LIN {X 0,Y 236.91,Z 434.305,A -85,B 0,C 180,E1 -22367.058,E2 -22367.058} C_VEL
LIN {X 0,Y 236.461,Z 436.627,A -85,B 0,C 180,E1 -22367.156,E2 -22367.156} C_VEL
LIN {X 0,Y 234.937,Z 442.325,A -85,B 0,C 180,E1 -22367.31,E2 -22367.31} C_VEL
LIN {X 0,Y 231.156,Z 451.531,A -85,B 0,C 180,E1 -22367.278,E2 -22367.278} C_VEL
LIN {X 0,Y 226.925,Z 460.5,A -85,B 0,C 180,E1 -22367.362,E2 -22367.362} C_VEL
LIN {X 0,Y 224.696,Z 465.695,A -85,B 0,C 180,E1 -22367.708,E2 -22367.708} C_VEL
LIN {X 0,Y 219.819,Z 477.382,A -85,B 0,C 180,E1 -22369.057,E2 -22369.057} C_VEL
LIN {X 0,Y 214.094,Z 488.851,A -85,B 0,C 180,E1 -22370.817,E2 -22370.817} C_VEL
LIN {X 0,Y 208.781,Z 498.232,A -85,B 0,C 180,E1 -22372.714,E2 -22372.714} C_VEL
LIN {X 0,Y 202.847,Z 507.555,A -85,B 0,C 180,E1 -22375.141,E2 -22375.141} C_VEL
LIN {X 0,Y 197.376,Z 515.201,A -85,B 0,C 180,E1 -22377.724,E2 -22377.724} C_VEL
LIN {X 0,Y 192.63,Z 521.438,A -85,B 0,C 180,E1 -22380.499,E2 -22380.499} C_VEL
LIN {X 0,Y 188.329,Z 526.526,A -85,B 0,C 180,E1 -22383.403,E2 -22383.403} C_VEL
LIN {X 0,Y 184.743,Z 530.596,A -85,B 0,C 180,E1 -22386.463,E2 -22386.463} C_VEL
LIN {X 0,Y 181.766,Z 533.709,A -85,B 0,C 180,E1 -22389.642,E2 -22389.642} C_VEL
LIN {X 0,Y 178.613,Z 536.431,A -85,B 0,C 180,E1 -22394.018,E2 -22394.018} C_VEL
LIN {X 0,Y 176.91,Z 537.692,A -85,B 0,C 180,E1 -22398.548,E2 -22398.548} C_VEL
LIN {X 0,Y 176.292,Z 537.397,A -85,B 0,C 180,E1 -22403.136,E2 -22403.136} C_VEL
LIN {X 0,Y 176.352,Z 536.677,A -85,B 0,C 180,E1 -22405.433,E2 -22405.433} C_VEL
LIN {X 0,Y 176.44,Z 535.538,A -85,B 0,C 180,E1 -22407.721,E2 -22407.721} C_VEL
LIN {X 0,Y 176.671,Z 533.977,A -85,B 0,C 180,E1 -22410.004,E2 -22410.004} C_VEL
LIN {X 0,Y 176.674,Z 530.644,A -85,B 0,C 180,E1 -22413.424,E2 -22413.424} C_VEL
LIN {X 0,Y 176.697,Z 527.213,A -85,B 0,C 180,E1 -22416.079,E2 -22416.079} C_VEL
LIN {X 0,Y 176.947,Z 521.277,A -85,B 0,C 180,E1 -22419.721,E2 -22419.721} C_VEL
LIN {X 0,Y 177.588,Z 514.102,A -85,B 0,C 180,E1 -22423.155,E2 -22423.155} C_VEL
LIN {X 0,Y 178.93,Z 505.14,A -85,B 0,C 180,E1 -22426.547,E2 -22426.547} C_VEL
LIN {X 0,Y 180.296,Z 495.891,A -85,B 0,C 180,E1 -22429.351,E2 -22429.351} C_VEL
LIN {X 0,Y 181.95,Z 485.894,A -85,B 0,C 180,E1 -22431.782,E2 -22431.782} C_VEL
LIN {X 0,Y 183.735,Z 474.492,A -85,B 0,C 180,E1 -22433.981,E2 -22433.981} C_VEL
LIN {X 0,Y 185.536,Z 462.13,A -85,B 0,C 180,E1 -22435.825,E2 -22435.825} C_VEL
LIN {X 0,Y 187.111,Z 449.244,A -85,B 0,C 180,E1 -22437.244,E2 -22437.244} C_VEL
LIN {X 0,Y 188.205,Z 437.063,A -85,B 0,C 180,E1 -22438.205,E2 -22438.205} C_VEL
LIN {X 0,Y 190.833,Z 387.8,A -85,B 0,C 180,E1 -22440.716,E2 -22440.716} C_VEL
LIN {X 0,Y 187.268,Z 349.514,A -85,B 0,C 180,E1 -22443.19,E2 -22443.19} C_VEL
LIN {X 0,Y 180.421,Z 327.475,A -85,B 0,C 180,E1 -22445.255,E2 -22445.255} C_VEL
LIN {X 0,Y 178.472,Z 318.252,A -85,B 0,C 180,E1 -22449.876,E2 -22449.876} C_VEL
LIN {X 0,Y 178.39,Z 318.26,A -85,B 0,C 180,E1 -22455.164,E2 -22455.164} C_VEL
LIN {X 0,Y 178.395,Z 318.261,A -85,B 0,C 180,E1 -22458.461,E2 -22458.461} C_VEL
LIN {X 0,Y 178.416,Z 318.259,A -85,B 0,C 180,E1 -22463.78,E2 -22463.78} C_VEL
LIN {X 0,Y 178.479,Z 318.252,A -85,B 0,C 180,E1 -22466.544,E2 -22466.544} C_VEL
LIN {X 0,Y 178.426,Z 318.258,A -85,B 0,C 180,E1 -22471.791,E2 -22471.791} C_VEL
LIN {X 0,Y 178.512,Z 318.249,A -85,B 0,C 180,E1 -22474.888,E2 -22474.888} C_VEL
LIN {X 0,Y 178.6,Z 318.237,A -85,B 0,C 180,E1 -22481.65,E2 -22481.65} C_VEL
LIN {X 0,Y 178.627,Z 318.23,A -85,B 0,C 180,E1 -22486.344,E2 -22486.344} C_VEL
LIN {X 0,Y 178.897,Z 318.2,A -85,B 0,C 180,E1 -22490.958,E2 -22490.958} C_VEL
LIN {X 0,Y 179.133,Z 318.171,A -85,B 0,C 180,E1 -22497.75,E2 -22497.75} C_VEL
LIN {X 0,Y 179.35,Z 318.142,A -85,B 0,C 180,E1 -22499.999,E2 -22499.999} C_VEL
LIN {X 0,Y 178.839,Z 318.205,A -85,B 0,C 180,E1 -22504.507,E2 -22504.507} C_VEL
LIN {X 0,Y 178.896,Z 318.199,A -85,B 0,C 180,E1 -22509.04,E2 -22509.04} C_VEL
LIN {X 0,Y 178.627,Z 318.235,A -85,B 0,C 180,E1 -22513.653,E2 -22513.653} C_VEL
LIN {X 0,Y 178.545,Z 318.239,A -85,B 0,C 180,E1 -22519.149,E2 -22519.149} C_VEL
LIN {X 0,Y 178.513,Z 318.247,A -85,B 0,C 180,E1 -22525.113,E2 -22525.113} C_VEL
LIN {X 0,Y 178.515,Z 318.249,A -85,B 0,C 180,E1 -22529.992,E2 -22529.992} C_VEL
LIN {X 0,Y 178.478,Z 318.25,A -85,B 0,C 180,E1 -22534.218,E2 -22534.218} C_VEL
LIN {X 0,Y 178.39,Z 318.262,A -85,B 0,C 180,E1 -22539.074,E2 -22539.074} C_VEL
LIN {X 0,Y 178.404,Z 318.261,A -85,B 0,C 180,E1 -22542.042,E2 -22542.042} C_VEL
LIN {X 0,Y 178.426,Z 318.254,A -85,B 0,C 180,E1 -22545.152,E2 -22545.152} C_VEL
LIN {X 0,Y 178.448,Z 318.257,A -85,B 0,C 180,E1 -22548.441,E2 -22548.441} C_VEL
LIN {X 0,Y 178.487,Z 318.249,A -85,B 0,C 180,E1 -22551.951,E2 -22551.951} C_VEL
LIN {X 0,Y 178.487,Z 318.252,A -85,B 0,C 180,E1 -22556.546,E2 -22556.546} C_VEL
LIN {X 0,Y 178.52,Z 318.246,A -85,B 0,C 180,E1 -22560.006,E2 -22560.006} C_VEL
LIN {X 0,Y 178.523,Z 318.247,A -85,B 0,C 180,E1 -22564.881,E2 -22564.881} C_VEL
LIN {X 0,Y 178.622,Z 318.233,A -85,B 0,C 180,E1 -22570.782,E2 -22570.782} C_VEL
LIN {X 0,Y 178.665,Z 318.228,A -85,B 0,C 180,E1 -22576.346,E2 -22576.346} C_VEL
LIN {X 0,Y 178.977,Z 318.19,A -85,B 0,C 180,E1 -22580.96,E2 -22580.96} C_VEL
LIN {X 0,Y 179.152,Z 318.165,A -85,B 0,C 180,E1 -22587.748,E2 -22587.748} C_VEL
LIN {X 0,Y 179.368,Z 318.141,A -85,B 0,C 180,E1 -22589.996,E2 -22589.996} C_VEL
LIN {X 0,Y 178.872,Z 318.201,A -85,B 0,C 180,E1 -22594.503,E2 -22594.503} C_VEL
LIN {X 0,Y 178.97,Z 318.192,A -85,B 0,C 180,E1 -22599.033,E2 -22599.033} C_VEL
LIN {X 0,Y 178.684,Z 318.226,A -85,B 0,C 180,E1 -22603.645,E2 -22603.645} C_VEL
LIN {X 0,Y 178.674,Z 318.227,A -85,B 0,C 180,E1 -22608.335,E2 -22608.335} C_VEL
LIN {X 0,Y 178.522,Z 318.248,A -85,B 0,C 180,E1 -22613.177,E2 -22613.177} C_VEL
LIN {X 0,Y 178.512,Z 318.249,A -85,B 0,C 180,E1 -22617.309,E2 -22617.309} C_VEL
LIN {X 0,Y 181.026,Z 325.006,A -85,B 0,C 180,E1 -22618.016,E2 -22618.016} C_VEL
LIN {X 0,Y 191.33,Z 351.912,A -85,B 0,C 180,E1 -22620.639,E2 -22620.639} C_VEL
LIN {X 0,Y 192.125,Z 354.048,A -85,B 0,C 180,E1 -22620.836,E2 -22620.836} C_VEL
LIN {X 0,Y 188.406,Z 416.37,A -85,B 0,C 180,E1 -22623.942,E2 -22623.942} C_VEL
LIN {X 0,Y 187.548,Z 428.759,A -85,B 0,C 180,E1 -22624.945,E2 -22624.945} C_VEL
LIN {X 0,Y 186.105,Z 441.894,A -85,B 0,C 180,E1 -22626.408,E2 -22626.408} C_VEL
LIN {X 0,Y 184.486,Z 453.979,A -85,B 0,C 180,E1 -22628.215,E2 -22628.215} C_VEL
LIN {X 0,Y 182.727,Z 466.025,A -85,B 0,C 180,E1 -22630.525,E2 -22630.525} C_VEL
LIN {X 0,Y 181.01,Z 476.642,A -85,B 0,C 180,E1 -22633.113,E2 -22633.113} C_VEL
LIN {X 0,Y 179.505,Z 486.117,A -85,B 0,C 180,E1 -22635.979,E2 -22635.979} C_VEL
LIN {X 0,Y 178.24,Z 494.278,A -85,B 0,C 180,E1 -22639.015,E2 -22639.015} C_VEL
LIN {X 0,Y 177.173,Z 501.741,A -85,B 0,C 180,E1 -22642.486,E2 -22642.486} C_VEL
LIN {X 0,Y 176.5,Z 507.92,A -85,B 0,C 180,E1 -22646.121,E2 -22646.121} C_VEL
LIN {X 0,Y 176.054,Z 513.063,A -85,B 0,C 180,E1 -22650.068,E2 -22650.068} C_VEL
LIN {X 0,Y 176.088,Z 516.711,A -85,B 0,C 180,E1 -22653.959,E2 -22653.959} C_VEL
LIN {X 0,Y 176.507,Z 518.42,A -85,B 0,C 180,E1 -22656.537,E2 -22656.537} C_VEL
LIN {X 0,Y 177.134,Z 519.648,A -85,B 0,C 180,E1 -22659.08,E2 -22659.08} C_VEL
LIN {X 0,Y 178.046,Z 520.342,A -85,B 0,C 180,E1 -22661.593,E2 -22661.593} C_VEL
LIN {X 0,Y 179.227,Z 520.555,A -85,B 0,C 180,E1 -22664.07,E2 -22664.07} C_VEL
LIN {X 0,Y 180.699,Z 520.318,A -85,B 0,C 180,E1 -22666.506,E2 -22666.506} C_VEL
LIN {X 0,Y 182.451,Z 519.566,A -85,B 0,C 180,E1 -22668.897,E2 -22668.897} C_VEL
LIN {X 0,Y 184.712,Z 518.19,A -85,B 0,C 180,E1 -22671.532,E2 -22671.532} C_VEL
LIN {X 0,Y 187.992,Z 515.646,A -85,B 0,C 180,E1 -22674.638,E2 -22674.638} C_VEL
LIN {X 0,Y 192.28,Z 511.728,A -85,B 0,C 180,E1 -22677.906,E2 -22677.906} C_VEL
LIN {X 0,Y 197.278,Z 506.305,A -85,B 0,C 180,E1 -22681.163,E2 -22681.163} C_VEL
LIN {X 0,Y 202.461,Z 499.893,A -85,B 0,C 180,E1 -22683.982,E2 -22683.982} C_VEL
LIN {X 0,Y 208.425,Z 491.476,A -85,B 0,C 180,E1 -22686.779,E2 -22686.779} C_VEL
LIN {X 0,Y 214.293,Z 481.83,A -85,B 0,C 180,E1 -22689.211,E2 -22689.211} C_VEL
LIN {X 0,Y 219.321,Z 472.21,A -85,B 0,C 180,E1 -22691.086,E2 -22691.086} C_VEL
LIN {X 0,Y 224.023,Z 461.664,A -85,B 0,C 180,E1 -22692.687,E2 -22692.687} C_VEL
LIN {X 0,Y 228.213,Z 450.32,A -85,B 0,C 180,E1 -22694.037,E2 -22694.037} C_VEL
LIN {X 0,Y 231.893,Z 438.008,A -85,B 0,C 180,E1 -22695.155,E2 -22695.155} C_VEL
LIN {X 0,Y 234.808,Z 424.844,A -85,B 0,C 180,E1 -22696.021,E2 -22696.021} C_VEL
LIN {X 0,Y 237.683,Z 405.575,A -85,B 0,C 180,E1 -22696.846,E2 -22696.846} C_VEL
LIN {X 0,Y 239.653,Z 391.45,A -85,B 0,C 180,E1 -22697.393,E2 -22697.393} C_VEL
LIN {X 0,Y 236.976,Z 385.819,A -85,B 0,C 180,E1 -22700.059,E2 -22700.059} C_VEL
LIN {X 0,Y 235.295,Z 382.982,A -85,B 0,C 180,E1 -22702.06,E2 -22702.06} C_VEL
LIN {X 0,Y 234.145,Z 380.911,A -85,B 0,C 180,E1 -22703.778,E2 -22703.778} C_VEL
LIN {X 0,Y 232.449,Z 378.806,A -85,B 0,C 180,E1 -22707.56,E2 -22707.56} C_VEL
LIN {X 0,Y 232.17,Z 378.586,A -85,B 0,C 180,E1 -22708.97,E2 -22708.97} C_VEL
LIN {X 0,Y 232.07,Z 379.141,A -85,B 0,C 180,E1 -22712.025,E2 -22712.025} C_VEL
LIN {X 0,Y 232.263,Z 379.966,A -85,B 0,C 180,E1 -22713.548,E2 -22713.548} C_VEL
LIN {X 0,Y 233.683,Z 384.466,A -85,B 0,C 180,E1 -22717.461,E2 -22717.461} C_VEL
LIN {X 0,Y 235.599,Z 389.873,A -85,B 0,C 180,E1 -22720.459,E2 -22720.459} C_VEL
LIN {X 0,Y 237.273,Z 395.332,A -85,B 0,C 180,E1 -22722.542,E2 -22722.542} C_VEL
LIN {X 0,Y 238.737,Z 400.557,A -85,B 0,C 180,E1 -22724.133,E2 -22724.133} C_VEL
LIN {X 0,Y 234.037,Z 433.293,A -85,B 0,C 180,E1 -22725.453,E2 -22725.453} C_VEL
LIN {X 0,Y 231.248,Z 445.622,A -85,B 0,C 180,E1 -22726.117,E2 -22726.117} C_VEL
LIN {X 0,Y 227.754,Z 457.295,A -85,B 0,C 180,E1 -22726.952,E2 -22726.952} C_VEL
LIN {X 0,Y 224.696,Z 465.695,A -85,B 0,C 180,E1 -22727.708,E2 -22727.708} C_VEL
LIN {X 0,Y 222.306,Z 470.885,A -85,B 0,C 180,E1 -22728.108,E2 -22728.108} C_VEL
LIN {X 0,Y 217.101,Z 479.22,A -85,B 0,C 180,E1 -22728.492,E2 -22728.492} C_VEL
LIN {X 0,Y 211.532,Z 487.12,A -85,B 0,C 180,E1 -22729.028,E2 -22729.028} C_VEL
LIN {X 0,Y 208.601,Z 491.616,A -85,B 0,C 180,E1 -22729.68,E2 -22729.68} C_VEL
LIN {X 0,Y 202.28,Z 501.788,A -85,B 0,C 180,E1 -22731.933,E2 -22731.933} C_VEL
LIN {X 0,Y 196.179,Z 510.356,A -85,B 0,C 180,E1 -22734.406,E2 -22734.406} C_VEL
LIN {X 0,Y 189.822,Z 518.369,A -85,B 0,C 180,E1 -22737.538,E2 -22737.538} C_VEL
LIN {X 0,Y 184.917,Z 523.953,A -85,B 0,C 180,E1 -22740.398,E2 -22740.398} C_VEL
LIN {X 0,Y 180.649,Z 528.482,A -85,B 0,C 180,E1 -22743.485,E2 -22743.485} C_VEL
LIN {X 0,Y 177.137,Z 531.918,A -85,B 0,C 180,E1 -22746.631,E2 -22746.631} C_VEL
LIN {X 0,Y 173.311,Z 535.193,A -85,B 0,C 180,E1 -22751.076,E2 -22751.076} C_VEL
LIN {X 0,Y 171.784,Z 536.265,A -85,B 0,C 180,E1 -22753.364,E2 -22753.364} C_VEL
LIN {X 0,Y 169.936,Z 537.251,A -85,B 0,C 180,E1 -22758.071,E2 -22758.071} C_VEL
LIN {X 0,Y 169.256,Z 536.745,A -85,B 0,C 180,E1 -22762.849,E2 -22762.849} C_VEL
LIN {X 0,Y 169.298,Z 535.932,A -85,B 0,C 180,E1 -22765.242,E2 -22765.242} C_VEL
LIN {X 0,Y 169.388,Z 534.689,A -85,B 0,C 180,E1 -22767.626,E2 -22767.626} C_VEL
LIN {X 0,Y 169.653,Z 532.994,A -85,B 0,C 180,E1 -22770.004,E2 -22770.004} C_VEL
LIN {X 0,Y 169.65,Z 529.491,A -85,B 0,C 180,E1 -22773.566,E2 -22773.566} C_VEL
LIN {X 0,Y 169.683,Z 524.72,A -85,B 0,C 180,E1 -22777.141,E2 -22777.141} C_VEL
LIN {X 0,Y 170.031,Z 518.573,A -85,B 0,C 180,E1 -22780.722,E2 -22780.722} C_VEL
LIN {X 0,Y 170.91,Z 510.862,A -85,B 0,C 180,E1 -22784.286,E2 -22784.286} C_VEL
LIN {X 0,Y 172.375,Z 501.133,A -85,B 0,C 180,E1 -22787.808,E2 -22787.808} C_VEL
LIN {X 0,Y 174.04,Z 491.112,A -85,B 0,C 180,E1 -22790.693,E2 -22790.693} C_VEL
LIN {X 0,Y 175.831,Z 480.218,A -85,B 0,C 180,E1 -22793.171,E2 -22793.171} C_VEL
LIN {X 0,Y 177.528,Z 469.019,A -85,B 0,C 180,E1 -22795.188,E2 -22795.188} C_VEL
LIN {X 0,Y 179.35,Z 456.267,A -85,B 0,C 180,E1 -22796.943,E2 -22796.943} C_VEL
LIN {X 0,Y 180.901,Z 442.079,A -85,B 0,C 180,E1 -22798.341,E2 -22798.341} C_VEL
LIN {X 0,Y 181.859,Z 427.344,A -85,B 0,C 180,E1 -22799.283,E2 -22799.283} C_VEL
LIN {X 0,Y 184.052,Z 388.689,A -85,B 0,C 180,E1 -22801.298,E2 -22801.298} C_VEL
LIN {X 0,Y 180.728,Z 351.595,A -85,B 0,C 180,E1 -22803.762,E2 -22803.762} C_VEL
LIN {X 0,Y 173.088,Z 327.033,A -85,B 0,C 180,E1 -22806.198,E2 -22806.198} C_VEL
LIN {X 0,Y 171.422,Z 319.131,A -85,B 0,C 180,E1 -22810.414,E2 -22810.414} C_VEL
LIN {X 0,Y 171.317,Z 319.139,A -85,B 0,C 180,E1 -22815.78,E2 -22815.78} C_VEL
LIN {X 0,Y 171.341,Z 319.141,A -85,B 0,C 180,E1 -22821.198,E2 -22821.198} C_VEL
LIN {X 0,Y 171.396,Z 319.136,A -85,B 0,C 180,E1 -22825.092,E2 -22825.092} C_VEL
LIN {X 0,Y 171.391,Z 319.135,A -85,B 0,C 180,E1 -22830.522,E2 -22830.522} C_VEL
LIN {X 0,Y 171.431,Z 319.126,A -85,B 0,C 180,E1 -22835.796,E2 -22835.796} C_VEL
LIN {X 0,Y 171.501,Z 319.122,A -85,B 0,C 180,E1 -22840.861,E2 -22840.861} C_VEL
LIN {X 0,Y 171.542,Z 319.113,A -85,B 0,C 180,E1 -22845.769,E2 -22845.769} C_VEL
LIN {X 0,Y 171.836,Z 319.079,A -85,B 0,C 180,E1 -22850.583,E2 -22850.583} C_VEL
LIN {X 0,Y 171.79,Z 319.083,A -85,B 0,C 180,E1 -22855.306,E2 -22855.306} C_VEL
LIN {X 0,Y 172.314,Z 319.018,A -85,B 0,C 180,E1 -22859.999,E2 -22859.999} C_VEL
LIN {X 0,Y 171.788,Z 319.084,A -85,B 0,C 180,E1 -22864.692,E2 -22864.692} C_VEL
LIN {X 0,Y 171.834,Z 319.078,A -85,B 0,C 180,E1 -22869.415,E2 -22869.415} C_VEL
LIN {X 0,Y 171.541,Z 319.116,A -85,B 0,C 180,E1 -22874.229,E2 -22874.229} C_VEL
LIN {X 0,Y 171.471,Z 319.121,A -85,B 0,C 180,E1 -22879.497,E2 -22879.497} C_VEL
LIN {X 0,Y 171.451,Z 319.128,A -85,B 0,C 180,E1 -22885.607,E2 -22885.607} C_VEL
LIN {X 0,Y 171.434,Z 319.129,A -85,B 0,C 180,E1 -22890.584,E2 -22890.584} C_VEL
LIN {X 0,Y 171.388,Z 319.132,A -85,B 0,C 180,E1 -22895.034,E2 -22895.034} C_VEL
LIN {X 0,Y 171.352,Z 319.139,A -85,B 0,C 180,E1 -22898.806,E2 -22898.806} C_VEL
LIN {X 0,Y 171.341,Z 319.138,A -85,B 0,C 180,E1 -22904.209,E2 -22904.209} C_VEL
LIN {X 0,Y 171.38,Z 319.136,A -85,B 0,C 180,E1 -22908.994,E2 -22908.994} C_VEL
LIN {X 0,Y 171.434,Z 319.127,A -85,B 0,C 180,E1 -22912.053,E2 -22912.053} C_VEL
LIN {X 0,Y 171.416,Z 319.132,A -85,B 0,C 180,E1 -22917.791,E2 -22917.791} C_VEL
LIN {X 0,Y 171.446,Z 319.124,A -85,B 0,C 180,E1 -22920.533,E2 -22920.533} C_VEL
LIN {X 0,Y 171.452,Z 319.128,A -85,B 0,C 180,E1 -22925.799,E2 -22925.799} C_VEL
LIN {X 0,Y 171.578,Z 319.11,A -85,B 0,C 180,E1 -22930.87,E2 -22930.87} C_VEL
LIN {X 0,Y 171.581,Z 319.11,A -85,B 0,C 180,E1 -22935.771,E2 -22935.771} C_VEL
LIN {X 0,Y 171.903,Z 319.072,A -85,B 0,C 180,E1 -22940.585,E2 -22940.585} C_VEL
LIN {X 0,Y 171.823,Z 319.077,A -85,B 0,C 180,E1 -22945.304,E2 -22945.304} C_VEL
LIN {X 0,Y 172.331,Z 319.017,A -85,B 0,C 180,E1 -22949.996,E2 -22949.996} C_VEL
LIN {X 0,Y 171.821,Z 319.079,A -85,B 0,C 180,E1 -22954.688,E2 -22954.688} C_VEL
LIN {X 0,Y 171.903,Z 319.071,A -85,B 0,C 180,E1 -22959.407,E2 -22959.407} C_VEL
LIN {X 0,Y 171.609,Z 319.108,A -85,B 0,C 180,E1 -22964.219,E2 -22964.219} C_VEL
LIN {X 0,Y 171.568,Z 319.115,A -85,B 0,C 180,E1 -22969.587,E2 -22969.587} C_VEL
LIN {X 0,Y 171.458,Z 319.126,A -85,B 0,C 180,E1 -22976.082,E2 -22976.082} C_VEL
LIN {X 0,Y 171.471,Z 319.125,A -85,B 0,C 180,E1 -22976.435,E2 -22976.435} C_VEL
LIN {X 0,Y 173.945,Z 325.721,A -85,B 0,C 180,E1 -22977.198,E2 -22977.198} C_VEL
LIN {X 0,Y 184.799,Z 354.048,A -85,B 0,C 180,E1 -22980.101,E2 -22980.101} C_VEL
LIN {X 0,Y 185.267,Z 355.43,A -85,B 0,C 180,E1 -22980.227,E2 -22980.227} C_VEL
LIN {X 0,Y 181.522,Z 416.426,A -85,B 0,C 180,E1 -22983.403,E2 -22983.403} C_VEL
LIN {X 0,Y 180.597,Z 429.111,A -85,B 0,C 180,E1 -22984.462,E2 -22984.462} C_VEL
LIN {X 0,Y 179.185,Z 441.892,A -85,B 0,C 180,E1 -22985.932,E2 -22985.932} C_VEL
LIN {X 0,Y 177.61,Z 453.393,A -85,B 0,C 180,E1 -22987.686,E2 -22987.686} C_VEL
LIN {X 0,Y 175.785,Z 465.628,A -85,B 0,C 180,E1 -22990.084,E2 -22990.084} C_VEL
LIN {X 0,Y 174.131,Z 475.694,A -85,B 0,C 180,E1 -22992.561,E2 -22992.561} C_VEL
LIN {X 0,Y 172.449,Z 485.991,A -85,B 0,C 180,E1 -22995.742,E2 -22995.742} C_VEL
LIN {X 0,Y 171.127,Z 494.299,A -85,B 0,C 180,E1 -22998.922,E2 -22998.922} C_VEL
LIN {X 0,Y 170.077,Z 501.686,A -85,B 0,C 180,E1 -23002.448,E2 -23002.448} C_VEL
LIN {X 0,Y 169.42,Z 507.657,A -85,B 0,C 180,E1 -23006.048,E2 -23006.048} C_VEL
LIN {X 0,Y 168.958,Z 512.818,A -85,B 0,C 180,E1 -23010.057,E2 -23010.057} C_VEL
LIN {X 0,Y 169,Z 516.675,A -85,B 0,C 180,E1 -23014.111,E2 -23014.111} C_VEL
LIN {X 0,Y 169.734,Z 519.274,A -85,B 0,C 180,E1 -23018.122,E2 -23018.122} C_VEL
LIN {X 0,Y 170.736,Z 520.456,A -85,B 0,C 180,E1 -23021.188,E2 -23021.188} C_VEL
LIN {X 0,Y 173.093,Z 521.034,A -85,B 0,C 180,E1 -23025.901,E2 -23025.901} C_VEL
LIN {X 0,Y 174.794,Z 520.643,A -85,B 0,C 180,E1 -23028.404,E2 -23028.404} C_VEL
LIN {X 0,Y 177.535,Z 519.411,A -85,B 0,C 180,E1 -23031.69,E2 -23031.69} C_VEL
LIN {X 0,Y 181.63,Z 516.694,A -85,B 0,C 180,E1 -23035.563,E2 -23035.563} C_VEL
LIN {X 0,Y 186.151,Z 513.001,A -85,B 0,C 180,E1 -23038.919,E2 -23038.919} C_VEL
LIN {X 0,Y 191.159,Z 508.078,A -85,B 0,C 180,E1 -23042.108,E2 -23042.108} C_VEL
LIN {X 0,Y 196.596,Z 502.036,A -85,B 0,C 180,E1 -23044.991,E2 -23044.991} C_VEL
LIN {X 0,Y 202.025,Z 495.155,A -85,B 0,C 180,E1 -23047.497,E2 -23047.497} C_VEL
LIN {X 0,Y 207.487,Z 487.165,A -85,B 0,C 180,E1 -23049.752,E2 -23049.752} C_VEL
LIN {X 0,Y 213.425,Z 477.159,A -85,B 0,C 180,E1 -23051.926,E2 -23051.926} C_VEL
LIN {X 0,Y 218.797,Z 466.528,A -85,B 0,C 180,E1 -23053.735,E2 -23053.735} C_VEL
LIN {X 0,Y 223.773,Z 454.668,A -85,B 0,C 180,E1 -23055.252,E2 -23055.252} C_VEL
LIN {X 0,Y 227.653,Z 443.2,A -85,B 0,C 180,E1 -23056.386,E2 -23056.386} C_VEL
LIN {X 0,Y 231.036,Z 430.008,A -85,B 0,C 180,E1 -23057.355,E2 -23057.355} C_VEL
LIN {X 0,Y 233.552,Z 416.586,A -85,B 0,C 180,E1 -23058.024,E2 -23058.024} C_VEL
LIN {X 0,Y 236.592,Z 395.886,A -85,B 0,C 180,E1 -23058.83,E2 -23058.83} C_VEL
LIN {X 0,Y 234.563,Z 391.349,A -85,B 0,C 180,E1 -23061.148,E2 -23061.148} C_VEL
LIN {X 0,Y 232.528,Z 387.703,A -85,B 0,C 180,E1 -23064.144,E2 -23064.144} C_VEL
LIN {X 0,Y 231.061,Z 385.742,A -85,B 0,C 180,E1 -23067.74,E2 -23067.74} C_VEL
LIN {X 0,Y 230.625,Z 385.684,A -85,B 0,C 180,E1 -23070.351,E2 -23070.351} C_VEL
LIN {X 0,Y 230.844,Z 386.618,A -85,B 0,C 180,E1 -23073.041,E2 -23073.041} C_VEL
LIN {X 0,Y 232.068,Z 391.278,A -85,B 0,C 180,E1 -23077.127,E2 -23077.127} C_VEL
LIN {X 0,Y 233.801,Z 396.999,A -85,B 0,C 180,E1 -23080.147,E2 -23080.147} C_VEL
LIN {X 0,Y 235.45,Z 402.957,A -85,B 0,C 180,E1 -23082.335,E2 -23082.335} C_VEL
LIN {X 0,Y 235.725,Z 404.141,A -85,B 0,C 180,E1 -23082.701,E2 -23082.701} C_VEL
LIN {X 0,Y 231.183,Z 433.416,A -85,B 0,C 180,E1 -23083.84,E2 -23083.84} C_VEL
LIN {X 0,Y 227.944,Z 446.952,A -85,B 0,C 180,E1 -23084.583,E2 -23084.583} C_VEL
LIN {X 0,Y 223.445,Z 460.592,A -85,B 0,C 180,E1 -23085.597,E2 -23085.597} C_VEL
LIN {X 0,Y 218.352,Z 472.911,A -85,B 0,C 180,E1 -23086.855,E2 -23086.855} C_VEL
LIN {X 0,Y 212.89,Z 483.97,A -85,B 0,C 180,E1 -23088.375,E2 -23088.375} C_VEL
LIN {X 0,Y 208.601,Z 491.616,A -85,B 0,C 180,E1 -23089.68,E2 -23089.68} C_VEL
LIN {X 0,Y 205.55,Z 496.055,A -85,B 0,C 180,E1 -23090.414,E2 -23090.414} C_VEL
LIN {X 0,Y 199.264,Z 503.034,A -85,B 0,C 180,E1 -23091.379,E2 -23091.379} C_VEL
LIN {X 0,Y 192.861,Z 509.347,A -85,B 0,C 180,E1 -23092.533,E2 -23092.533} C_VEL
LIN {X 0,Y 189.682,Z 512.773,A -85,B 0,C 180,E1 -23093.561,E2 -23093.561} C_VEL
LIN {X 0,Y 183.937,Z 519.376,A -85,B 0,C 180,E1 -23096.364,E2 -23096.364} C_VEL
LIN {X 0,Y 177.234,Z 526.128,A -85,B 0,C 180,E1 -23100.293,E2 -23100.293} C_VEL
LIN {X 0,Y 173.05,Z 530.026,A -85,B 0,C 180,E1 -23103.472,E2 -23103.472} C_VEL
LIN {X 0,Y 168.473,Z 533.806,A -85,B 0,C 180,E1 -23107.955,E2 -23107.955} C_VEL
LIN {X 0,Y 164.985,Z 536.022,A -85,B 0,C 180,E1 -23112.657,E2 -23112.657} C_VEL
LIN {X 0,Y 162.981,Z 536.78,A -85,B 0,C 180,E1 -23117.554,E2 -23117.554} C_VEL
LIN {X 0,Y 162.207,Z 536.084,A -85,B 0,C 180,E1 -23122.536,E2 -23122.536} C_VEL
LIN {X 0,Y 162.256,Z 535.129,A -85,B 0,C 180,E1 -23125.035,E2 -23125.035} C_VEL
LIN {X 0,Y 162.363,Z 533.755,A -85,B 0,C 180,E1 -23127.523,E2 -23127.523} C_VEL
LIN {X 0,Y 162.632,Z 531.961,A -85,B 0,C 180,E1 -23130.004,E2 -23130.004} C_VEL
LIN {X 0,Y 162.625,Z 528.257,A -85,B 0,C 180,E1 -23133.72,E2 -23133.72} C_VEL
LIN {X 0,Y 162.647,Z 523.289,A -85,B 0,C 180,E1 -23137.451,E2 -23137.451} C_VEL
LIN {X 0,Y 163.074,Z 516.935,A -85,B 0,C 180,E1 -23141.185,E2 -23141.185} C_VEL
LIN {X 0,Y 164.027,Z 508.866,A -85,B 0,C 180,E1 -23144.899,E2 -23144.899} C_VEL
LIN {X 0,Y 165.311,Z 500.616,A -85,B 0,C 180,E1 -23147.954,E2 -23147.954} C_VEL
LIN {X 0,Y 167.019,Z 490.572,A -85,B 0,C 180,E1 -23150.959,E2 -23150.959} C_VEL
LIN {X 0,Y 168.887,Z 479.464,A -85,B 0,C 180,E1 -23153.573,E2 -23153.573} C_VEL
LIN {X 0,Y 170.589,Z 468.405,A -85,B 0,C 180,E1 -23155.633,E2 -23155.633} C_VEL
LIN {X 0,Y 172.458,Z 455.574,A -85,B 0,C 180,E1 -23157.453,E2 -23157.453} C_VEL
LIN {X 0,Y 174.054,Z 441.322,A -85,B 0,C 180,E1 -23158.901,E2 -23158.901} C_VEL
LIN {X 0,Y 175.115,Z 425.135,A -85,B 0,C 180,E1 -23159.945,E2 -23159.945} C_VEL
LIN {X 0,Y 177.2,Z 388.779,A -85,B 0,C 180,E1 -23161.921,E2 -23161.921} C_VEL
LIN {X 0,Y 174.004,Z 353.186,A -85,B 0,C 180,E1 -23164.406,E2 -23164.406} C_VEL
LIN {X 0,Y 166.466,Z 329.072,A -85,B 0,C 180,E1 -23166.858,E2 -23166.858} C_VEL
LIN {X 0,Y 165.805,Z 326.738,A -85,B 0,C 180,E1 -23167.115,E2 -23167.115} C_VEL
LIN {X 0,Y 164.367,Z 320.011,A -85,B 0,C 180,E1 -23170.893,E2 -23170.893} C_VEL
LIN {X 0,Y 164.259,Z 320.019,A -85,B 0,C 180,E1 -23176.796,E2 -23176.796} C_VEL
LIN {X 0,Y 164.288,Z 320.021,A -85,B 0,C 180,E1 -23180.354,E2 -23180.354} C_VEL
LIN {X 0,Y 164.324,Z 320.015,A -85,B 0,C 180,E1 -23184.351,E2 -23184.351} C_VEL
LIN {X 0,Y 164.353,Z 320.013,A -85,B 0,C 180,E1 -23189.126,E2 -23189.126} C_VEL
LIN {X 0,Y 164.389,Z 320.007,A -85,B 0,C 180,E1 -23194.688,E2 -23194.688} C_VEL
LIN {X 0,Y 164.413,Z 320.003,A -85,B 0,C 180,E1 -23200.117,E2 -23200.117} C_VEL
LIN {X 0,Y 164.471,Z 319.994,A -85,B 0,C 180,E1 -23205.143,E2 -23205.143} C_VEL
LIN {X 0,Y 164.757,Z 319.961,A -85,B 0,C 180,E1 -23210.175,E2 -23210.175} C_VEL
LIN {X 0,Y 164.815,Z 319.952,A -85,B 0,C 180,E1 -23212.649,E2 -23212.649} C_VEL
LIN {X 0,Y 165.029,Z 319.929,A -85,B 0,C 180,E1 -23217.558,E2 -23217.558} C_VEL
LIN {X 0,Y 165.277,Z 319.895,A -85,B 0,C 180,E1 -23219.999,E2 -23219.999} C_VEL
LIN {X 0,Y 164.738,Z 319.962,A -85,B 0,C 180,E1 -23224.893,E2 -23224.893} C_VEL
LIN {X 0,Y 164.813,Z 319.956,A -85,B 0,C 180,E1 -23227.349,E2 -23227.349} C_VEL
LIN {X 0,Y 164.695,Z 319.964,A -85,B 0,C 180,E1 -23231.054,E2 -23231.054} C_VEL
LIN {X 0,Y 164.424,Z 320.003,A -85,B 0,C 180,E1 -23237.408,E2 -23237.408} C_VEL
LIN {X 0,Y 164.414,Z 320.002,A -85,B 0,C 180,E1 -23239.995,E2 -23239.995} C_VEL
LIN {X 0,Y 164.379,Z 320.005,A -85,B 0,C 180,E1 -23246.126,E2 -23246.126} C_VEL
LIN {X 0,Y 164.368,Z 320.009,A -85,B 0,C 180,E1 -23251.225,E2 -23251.225} C_VEL
LIN {X 0,Y 164.289,Z 320.016,A -85,B 0,C 180,E1 -23256.789,E2 -23256.789} C_VEL
LIN {X 0,Y 164.288,Z 320.022,A -85,B 0,C 180,E1 -23259.915,E2 -23259.915} C_VEL
LIN {X 0,Y 164.277,Z 320.018,A -85,B 0,C 180,E1 -23263.341,E2 -23263.341} C_VEL
LIN {X 0,Y 164.319,Z 320.015,A -85,B 0,C 180,E1 -23266.817,E2 -23266.817} C_VEL
LIN {X 0,Y 164.342,Z 320.012,A -85,B 0,C 180,E1 -23270.33,E2 -23270.33} C_VEL
LIN {X 0,Y 164.342,Z 320.012,A -85,B 0,C 180,E1 -23274.341,E2 -23274.341} C_VEL
LIN {X 0,Y 164.387,Z 320.005,A -85,B 0,C 180,E1 -23279.133,E2 -23279.133} C_VEL
LIN {X 0,Y 164.409,Z 320.005,A -85,B 0,C 180,E1 -23284.691,E2 -23284.691} C_VEL
LIN {X 0,Y 164.484,Z 319.991,A -85,B 0,C 180,E1 -23290.049,E2 -23290.049} C_VEL
LIN {X 0,Y 164.527,Z 319.989,A -85,B 0,C 180,E1 -23295.147,E2 -23295.147} C_VEL
LIN {X 0,Y 164.833,Z 319.951,A -85,B 0,C 180,E1 -23300.177,E2 -23300.177} C_VEL
LIN {X 0,Y 164.86,Z 319.95,A -85,B 0,C 180,E1 -23302.649,E2 -23302.649} C_VEL
LIN {X 0,Y 165.048,Z 319.922,A -85,B 0,C 180,E1 -23307.556,E2 -23307.556} C_VEL
LIN {X 0,Y 165.293,Z 319.894,A -85,B 0,C 180,E1 -23309.996,E2 -23309.996} C_VEL
LIN {X 0,Y 164.771,Z 319.957,A -85,B 0,C 180,E1 -23314.889,E2 -23314.889} C_VEL
LIN {X 0,Y 164.846,Z 319.949,A -85,B 0,C 180,E1 -23319.814,E2 -23319.814} C_VEL
LIN {X 0,Y 164.555,Z 319.986,A -85,B 0,C 180,E1 -23324.842,E2 -23324.842} C_VEL
LIN {X 0,Y 164.512,Z 319.994,A -85,B 0,C 180,E1 -23329.978,E2 -23329.978} C_VEL
LIN {X 0,Y 164.425,Z 320.002,A -85,B 0,C 180,E1 -23335.598,E2 -23335.598} C_VEL
LIN {X 0,Y 167.1,Z 327.088,A -85,B 0,C 180,E1 -23336.415,E2 -23336.415} C_VEL
LIN {X 0,Y 177.386,Z 353.948,A -85,B 0,C 180,E1 -23339.312,E2 -23339.312} C_VEL
LIN {X 0,Y 178.39,Z 356.628,A -85,B 0,C 180,E1 -23339.581,E2 -23339.581} C_VEL
LIN {X 0,Y 174.595,Z 417.374,A -85,B 0,C 180,E1 -23342.888,E2 -23342.888} C_VEL
LIN {X 0,Y 173.688,Z 429.269,A -85,B 0,C 180,E1 -23343.922,E2 -23343.922} C_VEL
LIN {X 0,Y 172.163,Z 442.671,A -85,B 0,C 180,E1 -23345.525,E2 -23345.525} C_VEL
LIN {X 0,Y 170.463,Z 454.766,A -85,B 0,C 180,E1 -23347.473,E2 -23347.473} C_VEL
LIN {X 0,Y 168.582,Z 466.976,A -85,B 0,C 180,E1 -23350.003,E2 -23350.003} C_VEL
LIN {X 0,Y 166.667,Z 478.396,A -85,B 0,C 180,E1 -23353.065,E2 -23353.065} C_VEL
LIN {X 0,Y 164.975,Z 488.274,A -85,B 0,C 180,E1 -23356.391,E2 -23356.391} C_VEL
LIN {X 0,Y 163.672,Z 496.568,A -85,B 0,C 180,E1 -23359.904,E2 -23359.904} C_VEL
LIN {X 0,Y 162.638,Z 504.546,A -85,B 0,C 180,E1 -23364.158,E2 -23364.158} C_VEL
LIN {X 0,Y 162.149,Z 509.054,A -85,B 0,C 180,E1 -23367.196,E2 -23367.196} C_VEL
LIN {X 0,Y 161.808,Z 514.093,A -85,B 0,C 180,E1 -23371.461,E2 -23371.461} C_VEL
LIN {X 0,Y 162.086,Z 517.604,A -85,B 0,C 180,E1 -23375.559,E2 -23375.559} C_VEL
LIN {X 0,Y 163.514,Z 520.5,A -85,B 0,C 180,E1 -23380.982,E2 -23380.982} C_VEL
LIN {X 0,Y 166.233,Z 521.504,A -85,B 0,C 180,E1 -23386.466,E2 -23386.466} C_VEL
LIN {X 0,Y 169.094,Z 520.969,A -85,B 0,C 180,E1 -23390.431,E2 -23390.431} C_VEL
LIN {X 0,Y 171.362,Z 520.056,A -85,B 0,C 180,E1 -23392.934,E2 -23392.934} C_VEL
LIN {X 0,Y 175.91,Z 517.357,A -85,B 0,C 180,E1 -23397.009,E2 -23397.009} C_VEL
LIN {X 0,Y 181.643,Z 512.959,A -85,B 0,C 180,E1 -23401.034,E2 -23401.034} C_VEL
LIN {X 0,Y 187.335,Z 507.759,A -85,B 0,C 180,E1 -23404.304,E2 -23404.304} C_VEL
LIN {X 0,Y 193.458,Z 501.151,A -85,B 0,C 180,E1 -23407.306,E2 -23407.306} C_VEL
LIN {X 0,Y 200.167,Z 492.8,A -85,B 0,C 180,E1 -23410.112,E2 -23410.112} C_VEL
LIN {X 0,Y 206.17,Z 484.108,A -85,B 0,C 180,E1 -23412.352,E2 -23412.352} C_VEL
LIN {X 0,Y 212.583,Z 473.167,A -85,B 0,C 180,E1 -23414.48,E2 -23414.48} C_VEL
LIN {X 0,Y 217.431,Z 463.356,A -85,B 0,C 180,E1 -23415.948,E2 -23415.948} C_VEL
LIN {X 0,Y 222.522,Z 450.934,A -85,B 0,C 180,E1 -23417.393,E2 -23417.393} C_VEL
LIN {X 0,Y 226.338,Z 439.302,A -85,B 0,C 180,E1 -23418.413,E2 -23418.413} C_VEL
LIN {X 0,Y 229.428,Z 426.853,A -85,B 0,C 180,E1 -23419.22,E2 -23419.22} C_VEL
LIN {X 0,Y 231.982,Z 411.938,A -85,B 0,C 180,E1 -23419.868,E2 -23419.868} C_VEL
LIN {X 0,Y 233.717,Z 400.237,A -85,B 0,C 180,E1 -23420.354,E2 -23420.354} C_VEL
LIN {X 0,Y 232.234,Z 396.865,A -85,B 0,C 180,E1 -23422.395,E2 -23422.395} C_VEL
LIN {X 0,Y 230.902,Z 394.42,A -85,B 0,C 180,E1 -23424.629,E2 -23424.629} C_VEL
LIN {X 0,Y 229.762,Z 392.779,A -85,B 0,C 180,E1 -23427.511,E2 -23427.511} C_VEL
LIN {X 0,Y 229.302,Z 392.623,A -85,B 0,C 180,E1 -23430.173,E2 -23430.173} C_VEL
LIN {X 0,Y 229.451,Z 393.502,A -85,B 0,C 180,E1 -23432.776,E2 -23432.776} C_VEL
LIN {X 0,Y 230.453,Z 398.012,A -85,B 0,C 180,E1 -23436.728,E2 -23436.728} C_VEL
LIN {X 0,Y 231.862,Z 403.29,A -85,B 0,C 180,E1 -23439.488,E2 -23439.488} C_VEL
LIN {X 0,Y 232.926,Z 407.843,A -85,B 0,C 180,E1 -23441.181,E2 -23441.181} C_VEL
LIN {X 0,Y 228.821,Z 432.987,A -85,B 0,C 180,E1 -23442.157,E2 -23442.157} C_VEL
LIN {X 0,Y 225.692,Z 445.51,A -85,B 0,C 180,E1 -23442.811,E2 -23442.811} C_VEL
LIN {X 0,Y 221.297,Z 458.58,A -85,B 0,C 180,E1 -23443.749,E2 -23443.749} C_VEL
LIN {X 0,Y 215.97,Z 471.247,A -85,B 0,C 180,E1 -23444.955,E2 -23444.955} C_VEL
LIN {X 0,Y 210.252,Z 482.547,A -85,B 0,C 180,E1 -23446.425,E2 -23446.425} C_VEL
LIN {X 0,Y 203.594,Z 493.758,A -85,B 0,C 180,E1 -23448.365,E2 -23448.365} C_VEL
LIN {X 0,Y 196.865,Z 503.562,A -85,B 0,C 180,E1 -23450.688,E2 -23450.688} C_VEL
LIN {X 0,Y 190.536,Z 511.71,A -85,B 0,C 180,E1 -23453.183,E2 -23453.183} C_VEL
LIN {X 0,Y 189.682,Z 512.773,A -85,B 0,C 180,E1 -23453.561,E2 -23453.561} C_VEL
LIN {X 0,Y 186.451,Z 516.085,A -85,B 0,C 180,E1 -23454.686,E2 -23454.686} C_VEL
LIN {X 0,Y 176.996,Z 522.883,A -85,B 0,C 180,E1 -23457.083,E2 -23457.083} C_VEL
LIN {X 0,Y 172.011,Z 526.16,A -85,B 0,C 180,E1 -23458.78,E2 -23458.78} C_VEL
LIN {X 0,Y 170.112,Z 527.571,A -85,B 0,C 180,E1 -23459.825,E2 -23459.825} C_VEL
LIN {X 0,Y 166.724,Z 530.341,A -85,B 0,C 180,E1 -23462.382,E2 -23462.382} C_VEL
LIN {X 0,Y 161.896,Z 533.795,A -85,B 0,C 180,E1 -23467.009,E2 -23467.009} C_VEL
LIN {X 0,Y 158.218,Z 535.764,A -85,B 0,C 180,E1 -23471.89,E2 -23471.89} C_VEL
LIN {X 0,Y 156.883,Z 536.213,A -85,B 0,C 180,E1 -23474.414,E2 -23474.414} C_VEL
LIN {X 0,Y 155.448,Z 535.984,A -85,B 0,C 180,E1 -23479.586,E2 -23479.586} C_VEL
LIN {X 0,Y 155.217,Z 534.192,A -85,B 0,C 180,E1 -23484.97,E2 -23484.97} C_VEL
LIN {X 0,Y 155.335,Z 532.819,A -85,B 0,C 180,E1 -23487.411,E2 -23487.411} C_VEL
LIN {X 0,Y 155.61,Z 530.902,A -85,B 0,C 180,E1 -23490.004,E2 -23490.004} C_VEL
LIN {X 0,Y 155.596,Z 526.984,A -85,B 0,C 180,E1 -23493.889,E2 -23493.889} C_VEL
LIN {X 0,Y 155.703,Z 520.739,A -85,B 0,C 180,E1 -23498.439,E2 -23498.439} C_VEL
LIN {X 0,Y 156.272,Z 513.831,A -85,B 0,C 180,E1 -23502.338,E2 -23502.338} C_VEL
LIN {X 0,Y 157.436,Z 505.13,A -85,B 0,C 180,E1 -23506.203,E2 -23506.203} C_VEL
LIN {X 0,Y 158.852,Z 496.181,A -85,B 0,C 180,E1 -23509.381,E2 -23509.381} C_VEL
LIN {X 0,Y 160.601,Z 486.445,A -85,B 0,C 180,E1 -23512.177,E2 -23512.177} C_VEL
LIN {X 0,Y 162.488,Z 475.259,A -85,B 0,C 180,E1 -23514.726,E2 -23514.726} C_VEL
LIN {X 0,Y 164.215,Z 464.157,A -85,B 0,C 180,E1 -23516.705,E2 -23516.705} C_VEL
LIN {X 0,Y 166.013,Z 451.313,A -85,B 0,C 180,E1 -23518.443,E2 -23518.443} C_VEL
LIN {X 0,Y 167.429,Z 437.774,A -85,B 0,C 180,E1 -23519.726,E2 -23519.726} C_VEL
LIN {X 0,Y 169.092,Z 411.634,A -85,B 0,C 180,E1 -23521.302,E2 -23521.302} C_VEL
LIN {X 0,Y 170.35,Z 388.643,A -85,B 0,C 180,E1 -23522.61,E2 -23522.61} C_VEL
LIN {X 0,Y 167.476,Z 355.25,A -85,B 0,C 180,E1 -23525.05,E2 -23525.05} C_VEL
LIN {X 0,Y 160.246,Z 331.904,A -85,B 0,C 180,E1 -23527.499,E2 -23527.499} C_VEL
LIN {X 0,Y 158.472,Z 326.255,A -85,B 0,C 180,E1 -23528.192,E2 -23528.192} C_VEL
LIN {X 0,Y 157.293,Z 320.892,A -85,B 0,C 180,E1 -23531.349,E2 -23531.349} C_VEL
LIN {X 0,Y 157.189,Z 320.902,A -85,B 0,C 180,E1 -23537.88,E2 -23537.88} C_VEL
LIN {X 0,Y 157.257,Z 320.895,A -85,B 0,C 180,E1 -23543.555,E2 -23543.555} C_VEL
LIN {X 0,Y 157.272,Z 320.893,A -85,B 0,C 180,E1 -23548.107,E2 -23548.107} C_VEL
LIN {X 0,Y 157.308,Z 320.89,A -85,B 0,C 180,E1 -23553.462,E2 -23553.462} C_VEL
LIN {X 0,Y 157.357,Z 320.883,A -85,B 0,C 180,E1 -23559.701,E2 -23559.701} C_VEL
LIN {X 0,Y 157.405,Z 320.874,A -85,B 0,C 180,E1 -23564.46,E2 -23564.46} C_VEL
LIN {X 0,Y 157.68,Z 320.843,A -85,B 0,C 180,E1 -23569.729,E2 -23569.729} C_VEL
LIN {X 0,Y 157.753,Z 320.831,A -85,B 0,C 180,E1 -23572.318,E2 -23572.318} C_VEL
LIN {X 0,Y 158.241,Z 320.771,A -85,B 0,C 180,E1 -23579.999,E2 -23579.999} C_VEL
LIN {X 0,Y 157.751,Z 320.835,A -85,B 0,C 180,E1 -23587.679,E2 -23587.679} C_VEL
LIN {X 0,Y 157.624,Z 320.845,A -85,B 0,C 180,E1 -23591.219,E2 -23591.219} C_VEL
LIN {X 0,Y 157.403,Z 320.879,A -85,B 0,C 180,E1 -23595.538,E2 -23595.538} C_VEL
LIN {X 0,Y 157.304,Z 320.887,A -85,B 0,C 180,E1 -23600.941,E2 -23600.941} C_VEL
LIN {X 0,Y 157.306,Z 320.885,A -85,B 0,C 180,E1 -23606.68,E2 -23606.68} C_VEL
LIN {X 0,Y 157.27,Z 320.894,A -85,B 0,C 180,E1 -23612.427,E2 -23612.427} C_VEL
LIN {X 0,Y 157.263,Z 320.892,A -85,B 0,C 180,E1 -23616.448,E2 -23616.448} C_VEL
LIN {X 0,Y 157.208,Z 320.901,A -85,B 0,C 180,E1 -23622.11,E2 -23622.11} C_VEL
LIN {X 0,Y 157.239,Z 320.899,A -85,B 0,C 180,E1 -23627.898,E2 -23627.898} C_VEL
LIN {X 0,Y 157.32,Z 320.883,A -85,B 0,C 180,E1 -23633.523,E2 -23633.523} C_VEL
LIN {X 0,Y 157.292,Z 320.893,A -85,B 0,C 180,E1 -23638.095,E2 -23638.095} C_VEL
LIN {X 0,Y 157.315,Z 320.887,A -85,B 0,C 180,E1 -23643.463,E2 -23643.463} C_VEL
LIN {X 0,Y 157.393,Z 320.873,A -85,B 0,C 180,E1 -23649.666,E2 -23649.666} C_VEL
LIN {X 0,Y 157.455,Z 320.872,A -85,B 0,C 180,E1 -23654.463,E2 -23654.463} C_VEL
LIN {X 0,Y 157.748,Z 320.832,A -85,B 0,C 180,E1 -23659.731,E2 -23659.731} C_VEL
LIN {X 0,Y 157.819,Z 320.827,A -85,B 0,C 180,E1 -23662.319,E2 -23662.319} C_VEL
LIN {X 0,Y 158.256,Z 320.771,A -85,B 0,C 180,E1 -23669.996,E2 -23669.996} C_VEL
LIN {X 0,Y 157.817,Z 320.826,A -85,B 0,C 180,E1 -23677.673,E2 -23677.673} C_VEL
LIN {X 0,Y 157.7,Z 320.839,A -85,B 0,C 180,E1 -23681.357,E2 -23681.357} C_VEL
LIN {X 0,Y 157.483,Z 320.864,A -85,B 0,C 180,E1 -23685.525,E2 -23685.525} C_VEL
LIN {X 0,Y 157.407,Z 320.879,A -85,B 0,C 180,E1 -23690.921,E2 -23690.921} C_VEL
LIN {X 0,Y 157.328,Z 320.894,A -85,B 0,C 180,E1 -23694.663,E2 -23694.663} C_VEL
LIN {X 0,Y 160.92,Z 330.129,A -85,B 0,C 180,E1 -23695.802,E2 -23695.802} C_VEL
LIN {X 0,Y 171.098,Z 356.788,A -85,B 0,C 180,E1 -23698.774,E2 -23698.774} C_VEL
LIN {X 0,Y 171.614,Z 358.66,A -85,B 0,C 180,E1 -23698.951,E2 -23698.951} C_VEL
LIN {X 0,Y 167.76,Z 417.083,A -85,B 0,C 180,E1 -23702.253,E2 -23702.253} C_VEL
LIN {X 0,Y 166.826,Z 429.213,A -85,B 0,C 180,E1 -23703.342,E2 -23703.342} C_VEL
LIN {X 0,Y 165.22,Z 442.846,A -85,B 0,C 180,E1 -23705.033,E2 -23705.033} C_VEL
LIN {X 0,Y 163.402,Z 455.419,A -85,B 0,C 180,E1 -23707.154,E2 -23707.154} C_VEL
LIN {X 0,Y 161.553,Z 467.019,A -85,B 0,C 180,E1 -23709.666,E2 -23709.666} C_VEL
LIN {X 0,Y 159.761,Z 477.496,A -85,B 0,C 180,E1 -23712.539,E2 -23712.539} C_VEL
LIN {X 0,Y 158.085,Z 487.041,A -85,B 0,C 180,E1 -23715.793,E2 -23715.793} C_VEL
LIN {X 0,Y 156.885,Z 494.496,A -85,B 0,C 180,E1 -23718.905,E2 -23718.905} C_VEL
LIN {X 0,Y 155.863,Z 501.572,A -85,B 0,C 180,E1 -23722.504,E2 -23722.504} C_VEL
LIN {X 0,Y 155.284,Z 506.771,A -85,B 0,C 180,E1 -23725.745,E2 -23725.745} C_VEL
LIN {X 0,Y 154.776,Z 512.256,A -85,B 0,C 180,E1 -23730.036,E2 -23730.036} C_VEL
LIN {X 0,Y 154.927,Z 516.993,A -85,B 0,C 180,E1 -23735.108,E2 -23735.108} C_VEL
LIN {X 0,Y 155.657,Z 519.458,A -85,B 0,C 180,E1 -23738.827,E2 -23738.827} C_VEL
LIN {X 0,Y 156.615,Z 520.775,A -85,B 0,C 180,E1 -23741.694,E2 -23741.694} C_VEL
LIN {X 0,Y 158.991,Z 521.932,A -85,B 0,C 180,E1 -23746.485,E2 -23746.485} C_VEL
LIN {X 0,Y 161.393,Z 521.864,A -85,B 0,C 180,E1 -23749.97,E2 -23749.97} C_VEL
LIN {X 0,Y 163.667,Z 521.312,A -85,B 0,C 180,E1 -23752.6,E2 -23752.6} C_VEL
LIN {X 0,Y 166.217,Z 520.26,A -85,B 0,C 180,E1 -23755.15,E2 -23755.15} C_VEL
LIN {X 0,Y 169.095,Z 518.743,A -85,B 0,C 180,E1 -23757.619,E2 -23757.619} C_VEL
LIN {X 0,Y 174.09,Z 515.538,A -85,B 0,C 180,E1 -23761.159,E2 -23761.159} C_VEL
LIN {X 0,Y 179.631,Z 511.152,A -85,B 0,C 180,E1 -23764.489,E2 -23764.489} C_VEL
LIN {X 0,Y 186.006,Z 505.247,A -85,B 0,C 180,E1 -23767.65,E2 -23767.65} C_VEL
LIN {X 0,Y 193.039,Z 497.629,A -85,B 0,C 180,E1 -23770.631,E2 -23770.631} C_VEL
LIN {X 0,Y 200.042,Z 488.726,A -85,B 0,C 180,E1 -23773.202,E2 -23773.202} C_VEL
LIN {X 0,Y 206.698,Z 478.675,A -85,B 0,C 180,E1 -23775.382,E2 -23775.382} C_VEL
LIN {X 0,Y 212.447,Z 468.558,A -85,B 0,C 180,E1 -23777.074,E2 -23777.074} C_VEL
LIN {X 0,Y 217.647,Z 457.501,A -85,B 0,C 180,E1 -23778.494,E2 -23778.494} C_VEL
LIN {X 0,Y 222.46,Z 444.786,A -85,B 0,C 180,E1 -23779.734,E2 -23779.734} C_VEL
LIN {X 0,Y 226.358,Z 431.182,A -85,B 0,C 180,E1 -23780.7,E2 -23780.7} C_VEL
LIN {X 0,Y 228.934,Z 418.751,A -85,B 0,C 180,E1 -23781.313,E2 -23781.313} C_VEL
LIN {X 0,Y 231.131,Z 404.906,A -85,B 0,C 180,E1 -23781.883,E2 -23781.883} C_VEL
LIN {X 0,Y 229.55,Z 401.464,A -85,B 0,C 180,E1 -23784.582,E2 -23784.582} C_VEL
LIN {X 0,Y 228.277,Z 399.63,A -85,B 0,C 180,E1 -23788.101,E2 -23788.101} C_VEL
LIN {X 0,Y 227.945,Z 399.783,A -85,B 0,C 180,E1 -23791.099,E2 -23791.099} C_VEL
LIN {X 0,Y 228.043,Z 400.441,A -85,B 0,C 180,E1 -23792.51,E2 -23792.51} C_VEL
LIN {X 0,Y 228.809,Z 404.439,A -85,B 0,C 180,E1 -23796.112,E2 -23796.112} C_VEL
LIN {X 0,Y 229.962,Z 409.6,A -85,B 0,C 180,E1 -23798.817,E2 -23798.817} C_VEL
LIN {X 0,Y 230.314,Z 411.928,A -85,B 0,C 180,E1 -23799.65,E2 -23799.65} C_VEL
LIN {X 0,Y 226.457,Z 433.713,A -85,B 0,C 180,E1 -23800.481,E2 -23800.481} C_VEL
LIN {X 0,Y 222.903,Z 446.924,A -85,B 0,C 180,E1 -23801.181,E2 -23801.181} C_VEL
LIN {X 0,Y 218.021,Z 460.518,A -85,B 0,C 180,E1 -23802.159,E2 -23802.159} C_VEL
LIN {X 0,Y 212.531,Z 472.542,A -85,B 0,C 180,E1 -23803.333,E2 -23803.333} C_VEL
LIN {X 0,Y 206.604,Z 483.437,A -85,B 0,C 180,E1 -23804.767,E2 -23804.767} C_VEL
LIN {X 0,Y 199.696,Z 494.336,A -85,B 0,C 180,E1 -23806.674,E2 -23806.674} C_VEL
LIN {X 0,Y 192.688,Z 503.965,A -85,B 0,C 180,E1 -23808.974,E2 -23808.974} C_VEL
LIN {X 0,Y 186.052,Z 511.888,A -85,B 0,C 180,E1 -23811.453,E2 -23811.453} C_VEL
LIN {X 0,Y 179.942,Z 518.414,A -85,B 0,C 180,E1 -23814.145,E2 -23814.145} C_VEL
LIN {X 0,Y 174.532,Z 523.74,A -85,B 0,C 180,E1 -23817.078,E2 -23817.078} C_VEL
LIN {X 0,Y 170.112,Z 527.571,A -85,B 0,C 180,E1 -23819.825,E2 -23819.825} C_VEL
LIN {X 0,Y 167.189,Z 529.55,A -85,B 0,C 180,E1 -23821.442,E2 -23821.442} C_VEL
LIN {X 0,Y 161.071,Z 532.233,A -85,B 0,C 180,E1 -23824.003,E2 -23824.003} C_VEL
LIN {X 0,Y 155.304,Z 534.171,A -85,B 0,C 180,E1 -23826.83,E2 -23826.83} C_VEL
LIN {X 0,Y 153.006,Z 534.908,A -85,B 0,C 180,E1 -23828.828,E2 -23828.828} C_VEL
LIN {X 0,Y 150.031,Z 535.766,A -85,B 0,C 180,E1 -23833.683,E2 -23833.683} C_VEL
LIN {X 0,Y 148.477,Z 535.31,A -85,B 0,C 180,E1 -23839.091,E2 -23839.091} C_VEL
LIN {X 0,Y 148.182,Z 533.378,A -85,B 0,C 180,E1 -23844.562,E2 -23844.562} C_VEL
LIN {X 0,Y 148.412,Z 530.814,A -85,B 0,C 180,E1 -23848.648,E2 -23848.648} C_VEL
LIN {X 0,Y 148.526,Z 528.496,A -85,B 0,C 180,E1 -23851.36,E2 -23851.36} C_VEL
LIN {X 0,Y 148.564,Z 523.969,A -85,B 0,C 180,E1 -23855.433,E2 -23855.433} C_VEL
LIN {X 0,Y 148.76,Z 518.006,A -85,B 0,C 180,E1 -23859.521,E2 -23859.521} C_VEL
LIN {X 0,Y 149.488,Z 510.487,A -85,B 0,C 180,E1 -23863.599,E2 -23863.599} C_VEL
LIN {X 0,Y 150.692,Z 502.827,A -85,B 0,C 180,E1 -23866.95,E2 -23866.95} C_VEL
LIN {X 0,Y 152.2,Z 493.453,A -85,B 0,C 180,E1 -23870.265,E2 -23870.265} C_VEL
LIN {X 0,Y 154.291,Z 481.874,A -85,B 0,C 180,E1 -23873.491,E2 -23873.491} C_VEL
LIN {X 0,Y 156.168,Z 470.832,A -85,B 0,C 180,E1 -23875.9,E2 -23875.9} C_VEL
LIN {X 0,Y 158.259,Z 457.164,A -85,B 0,C 180,E1 -23878.155,E2 -23878.155} C_VEL
LIN {X 0,Y 159.894,Z 443.962,A -85,B 0,C 180,E1 -23879.728,E2 -23879.728} C_VEL
LIN {X 0,Y 160.952,Z 431.165,A -85,B 0,C 180,E1 -23880.778,E2 -23880.778} C_VEL
LIN {X 0,Y 163.57,Z 389.417,A -85,B 0,C 180,E1 -23883.275,E2 -23883.275} C_VEL
LIN {X 0,Y 160.765,Z 356.642,A -85,B 0,C 180,E1 -23885.758,E2 -23885.758} C_VEL
LIN {X 0,Y 153.369,Z 332.678,A -85,B 0,C 180,E1 -23888.419,E2 -23888.419} C_VEL
LIN {X 0,Y 151.132,Z 325.859,A -85,B 0,C 180,E1 -23889.31,E2 -23889.31} C_VEL
LIN {X 0,Y 150.228,Z 321.771,A -85,B 0,C 180,E1 -23891.825,E2 -23891.825} C_VEL
LIN {X 0,Y 150.128,Z 321.779,A -85,B 0,C 180,E1 -23895.394,E2 -23895.394} C_VEL
LIN {X 0,Y 150.136,Z 321.784,A -85,B 0,C 180,E1 -23899.052,E2 -23899.052} C_VEL
LIN {X 0,Y 150.175,Z 321.776,A -85,B 0,C 180,E1 -23902.709,E2 -23902.709} C_VEL
LIN {X 0,Y 150.2,Z 321.775,A -85,B 0,C 180,E1 -23907.376,E2 -23907.376} C_VEL
LIN {X 0,Y 150.226,Z 321.772,A -85,B 0,C 180,E1 -23912.73,E2 -23912.73} C_VEL
LIN {X 0,Y 150.281,Z 321.764,A -85,B 0,C 180,E1 -23919.276,E2 -23919.276} C_VEL
LIN {X 0,Y 150.31,Z 321.758,A -85,B 0,C 180,E1 -23923.706,E2 -23923.706} C_VEL
LIN {X 0,Y 150.601,Z 321.726,A -85,B 0,C 180,E1 -23929.24,E2 -23929.24} C_VEL
LIN {X 0,Y 150.676,Z 321.713,A -85,B 0,C 180,E1 -23931.955,E2 -23931.955} C_VEL
LIN {X 0,Y 151.202,Z 321.648,A -85,B 0,C 180,E1 -23939.999,E2 -23939.999} C_VEL
LIN {X 0,Y 150.674,Z 321.715,A -85,B 0,C 180,E1 -23948.043,E2 -23948.043} C_VEL
LIN {X 0,Y 150.567,Z 321.724,A -85,B 0,C 180,E1 -23951.423,E2 -23951.423} C_VEL
LIN {X 0,Y 150.308,Z 321.76,A -85,B 0,C 180,E1 -23956.291,E2 -23956.291} C_VEL
LIN {X 0,Y 150.279,Z 321.762,A -85,B 0,C 180,E1 -23960.722,E2 -23960.722} C_VEL
LIN {X 0,Y 150.237,Z 321.766,A -85,B 0,C 180,E1 -23967.278,E2 -23967.278} C_VEL
LIN {X 0,Y 150.21,Z 321.773,A -85,B 0,C 180,E1 -23972.63,E2 -23972.63} C_VEL
LIN {X 0,Y 150.169,Z 321.775,A -85,B 0,C 180,E1 -23977.473,E2 -23977.473} C_VEL
LIN {X 0,Y 150.147,Z 321.781,A -85,B 0,C 180,E1 -23981.503,E2 -23981.503} C_VEL
LIN {X 0,Y 150.14,Z 321.778,A -85,B 0,C 180,E1 -23985.4,E2 -23985.4} C_VEL
LIN {X 0,Y 150.188,Z 321.776,A -85,B 0,C 180,E1 -23989.07,E2 -23989.07} C_VEL
LIN {X 0,Y 150.229,Z 321.766,A -85,B 0,C 180,E1 -23992.681,E2 -23992.681} C_VEL
LIN {X 0,Y 150.215,Z 321.772,A -85,B 0,C 180,E1 -23997.365,E2 -23997.365} C_VEL
LIN {X 0,Y 150.24,Z 321.769,A -85,B 0,C 180,E1 -24002.719,E2 -24002.719} C_VEL
LIN {X 0,Y 150.35,Z 321.75,A -85,B 0,C 180,E1 -24009.206,E2 -24009.206} C_VEL
LIN {X 0,Y 150.362,Z 321.754,A -85,B 0,C 180,E1 -24013.711,E2 -24013.711} C_VEL
LIN {X 0,Y 150.662,Z 321.715,A -85,B 0,C 180,E1 -24019.243,E2 -24019.243} C_VEL
LIN {X 0,Y 150.755,Z 321.706,A -85,B 0,C 180,E1 -24021.957,E2 -24021.957} C_VEL
LIN {X 0,Y 151.216,Z 321.648,A -85,B 0,C 180,E1 -24029.996,E2 -24029.996} C_VEL
LIN {X 0,Y 150.756,Z 321.706,A -85,B 0,C 180,E1 -24038.034,E2 -24038.034} C_VEL
LIN {X 0,Y 150.629,Z 321.72,A -85,B 0,C 180,E1 -24041.54,E2 -24041.54} C_VEL
LIN {X 0,Y 150.391,Z 321.747,A -85,B 0,C 180,E1 -24046.277,E2 -24046.277} C_VEL
LIN {X 0,Y 150.381,Z 321.754,A -85,B 0,C 180,E1 -24050.826,E2 -24050.826} C_VEL
LIN {X 0,Y 150.265,Z 321.768,A -85,B 0,C 180,E1 -24053.601,E2 -24053.601} C_VEL
LIN {X 0,Y 152.144,Z 326.705,A -85,B 0,C 180,E1 -24054.286,E2 -24054.286} C_VEL
LIN {X 0,Y 160.64,Z 348.346,A -85,B 0,C 180,E1 -24056.987,E2 -24056.987} C_VEL
LIN {X 0,Y 164.72,Z 359.401,A -85,B 0,C 180,E1 -24058.215,E2 -24058.215} C_VEL
LIN {X 0,Y 160.9,Z 417.169,A -85,B 0,C 180,E1 -24061.64,E2 -24061.64} C_VEL
LIN {X 0,Y 159.981,Z 428.749,A -85,B 0,C 180,E1 -24062.701,E2 -24062.701} C_VEL
LIN {X 0,Y 158.383,Z 442.143,A -85,B 0,C 180,E1 -24064.399,E2 -24064.399} C_VEL
LIN {X 0,Y 156.803,Z 453.041,A -85,B 0,C 180,E1 -24066.221,E2 -24066.221} C_VEL
LIN {X 0,Y 155.023,Z 464.029,A -85,B 0,C 180,E1 -24068.555,E2 -24068.555} C_VEL
LIN {X 0,Y 152.975,Z 475.728,A -85,B 0,C 180,E1 -24071.709,E2 -24071.709} C_VEL
LIN {X 0,Y 151.366,Z 485.058,A -85,B 0,C 180,E1 -24074.857,E2 -24074.857} C_VEL
LIN {X 0,Y 149.862,Z 493.946,A -85,B 0,C 180,E1 -24078.607,E2 -24078.607} C_VEL
LIN {X 0,Y 148.691,Z 502.107,A -85,B 0,C 180,E1 -24082.932,E2 -24082.932} C_VEL
LIN {X 0,Y 148.038,Z 508.066,A -85,B 0,C 180,E1 -24086.912,E2 -24086.912} C_VEL
LIN {X 0,Y 147.625,Z 513.487,A -85,B 0,C 180,E1 -24091.572,E2 -24091.572} C_VEL
LIN {X 0,Y 147.969,Z 517.502,A -85,B 0,C 180,E1 -24096.191,E2 -24096.191} C_VEL
LIN {X 0,Y 149.119,Z 520.265,A -85,B 0,C 180,E1 -24100.738,E2 -24100.738} C_VEL
LIN {X 0,Y 150.28,Z 521.49,A -85,B 0,C 180,E1 -24103.706,E2 -24103.706} C_VEL
LIN {X 0,Y 151.812,Z 522.218,A -85,B 0,C 180,E1 -24106.618,E2 -24106.618} C_VEL
LIN {X 0,Y 153.683,Z 522.47,A -85,B 0,C 180,E1 -24109.461,E2 -24109.461} C_VEL
LIN {X 0,Y 155.986,Z 522.274,A -85,B 0,C 180,E1 -24112.325,E2 -24112.325} C_VEL
LIN {X 0,Y 158.478,Z 521.619,A -85,B 0,C 180,E1 -24114.913,E2 -24114.913} C_VEL
LIN {X 0,Y 161.732,Z 520.321,A -85,B 0,C 180,E1 -24117.83,E2 -24117.83} C_VEL
LIN {X 0,Y 166.346,Z 517.895,A -85,B 0,C 180,E1 -24121.212,E2 -24121.212} C_VEL
LIN {X 0,Y 171.982,Z 514.152,A -85,B 0,C 180,E1 -24124.689,E2 -24124.689} C_VEL
LIN {X 0,Y 178.803,Z 508.766,A -85,B 0,C 180,E1 -24128.151,E2 -24128.151} C_VEL
LIN {X 0,Y 186.345,Z 501.575,A -85,B 0,C 180,E1 -24131.354,E2 -24131.354} C_VEL
LIN {X 0,Y 194.056,Z 492.916,A -85,B 0,C 180,E1 -24134.151,E2 -24134.151} C_VEL
LIN {X 0,Y 200.648,Z 484.179,A -85,B 0,C 180,E1 -24136.274,E2 -24136.274} C_VEL
LIN {X 0,Y 206.999,Z 474.309,A -85,B 0,C 180,E1 -24138.102,E2 -24138.102} C_VEL
LIN {X 0,Y 213.191,Z 462.714,A -85,B 0,C 180,E1 -24139.75,E2 -24139.75} C_VEL
LIN {X 0,Y 218.275,Z 451.176,A -85,B 0,C 180,E1 -24140.998,E2 -24140.998} C_VEL
LIN {X 0,Y 222.652,Z 438.617,A -85,B 0,C 180,E1 -24142.003,E2 -24142.003} C_VEL
LIN {X 0,Y 225.877,Z 426.07,A -85,B 0,C 180,E1 -24142.74,E2 -24142.74} C_VEL
LIN {X 0,Y 228.722,Z 410.055,A -85,B 0,C 180,E1 -24143.409,E2 -24143.409} C_VEL
LIN {X 0,Y 227.832,Z 408.069,A -85,B 0,C 180,E1 -24145.291,E2 -24145.291} C_VEL
LIN {X 0,Y 227.007,Z 406.71,A -85,B 0,C 180,E1 -24147.672,E2 -24147.672} C_VEL
LIN {X 0,Y 226.562,Z 406.629,A -85,B 0,C 180,E1 -24150.524,E2 -24150.524} C_VEL
LIN {X 0,Y 226.648,Z 407.366,A -85,B 0,C 180,E1 -24152.263,E2 -24152.263} C_VEL
LIN {X 0,Y 227.192,Z 410.985,A -85,B 0,C 180,E1 -24155.532,E2 -24155.532} C_VEL
LIN {X 0,Y 228.049,Z 415.72,A -85,B 0,C 180,E1 -24158.052,E2 -24158.052} C_VEL
LIN {X 0,Y 224.643,Z 433.796,A -85,B 0,C 180,E1 -24158.728,E2 -24158.728} C_VEL
LIN {X 0,Y 221.051,Z 446.44,A -85,B 0,C 180,E1 -24159.383,E2 -24159.383} C_VEL
LIN {X 0,Y 216.337,Z 459.072,A -85,B 0,C 180,E1 -24160.244,E2 -24160.244} C_VEL
LIN {X 0,Y 210.666,Z 471.24,A -85,B 0,C 180,E1 -24161.367,E2 -24161.367} C_VEL
LIN {X 0,Y 203.838,Z 483.416,A -85,B 0,C 180,E1 -24162.901,E2 -24162.901} C_VEL
LIN {X 0,Y 197.285,Z 493.302,A -85,B 0,C 180,E1 -24164.574,E2 -24164.574} C_VEL
LIN {X 0,Y 189.854,Z 502.94,A -85,B 0,C 180,E1 -24166.788,E2 -24166.788} C_VEL
LIN {X 0,Y 182.887,Z 510.939,A -85,B 0,C 180,E1 -24169.221,E2 -24169.221} C_VEL
LIN {X 0,Y 176.387,Z 517.519,A -85,B 0,C 180,E1 -24171.869,E2 -24171.869} C_VEL
LIN {X 0,Y 170.458,Z 522.874,A -85,B 0,C 180,E1 -24174.754,E2 -24174.754} C_VEL
LIN {X 0,Y 163.873,Z 528.159,A -85,B 0,C 180,E1 -24178.687,E2 -24178.687} C_VEL
LIN {X 0,Y 160.471,Z 530.605,A -85,B 0,C 180,E1 -24181.208,E2 -24181.208} C_VEL
LIN {X 0,Y 155.373,Z 533.771,A -85,B 0,C 180,E1 -24185.984,E2 -24185.984} C_VEL
LIN {X 0,Y 153.006,Z 534.908,A -85,B 0,C 180,E1 -24188.828,E2 -24188.828} C_VEL
LIN {X 0,Y 150.919,Z 535.433,A -85,B 0,C 180,E1 -24190.907,E2 -24190.907} C_VEL
LIN {X 0,Y 146.287,Z 535.559,A -85,B 0,C 180,E1 -24194.29,E2 -24194.29} C_VEL
LIN {X 0,Y 142.926,Z 535.011,A -85,B 0,C 180,E1 -24197.132,E2 -24197.132} C_VEL
LIN {X 0,Y 141.448,Z 534.347,A -85,B 0,C 180,E1 -24199.422,E2 -24199.422} C_VEL
LIN {X 0,Y 141.275,Z 534.065,A -85,B 0,C 180,E1 -24200.211,E2 -24200.211} C_VEL
LIN {X 0,Y 141.192,Z 532.238,A -85,B 0,C 180,E1 -24204.592,E2 -24204.592} C_VEL
LIN {X 0,Y 141.434,Z 529.651,A -85,B 0,C 180,E1 -24208.581,E2 -24208.581} C_VEL
LIN {X 0,Y 141.552,Z 527.182,A -85,B 0,C 180,E1 -24211.427,E2 -24211.427} C_VEL
LIN {X 0,Y 141.569,Z 522.401,A -85,B 0,C 180,E1 -24215.702,E2 -24215.702} C_VEL
LIN {X 0,Y 141.786,Z 516.204,A -85,B 0,C 180,E1 -24219.994,E2 -24219.994} C_VEL
LIN {X 0,Y 142.442,Z 509.812,A -85,B 0,C 180,E1 -24223.557,E2 -24223.557} C_VEL
LIN {X 0,Y 143.656,Z 502.15,A -85,B 0,C 180,E1 -24227.073,E2 -24227.073} C_VEL
LIN {X 0,Y 145.368,Z 491.626,A -85,B 0,C 180,E1 -24230.891,E2 -24230.891} C_VEL
LIN {X 0,Y 147.345,Z 481.056,A -85,B 0,C 180,E1 -24233.92,E2 -24233.92} C_VEL
LIN {X 0,Y 149.207,Z 470.223,A -85,B 0,C 180,E1 -24236.371,E2 -24236.371} C_VEL
LIN {X 0,Y 151.271,Z 457.125,A -85,B 0,C 180,E1 -24238.629,E2 -24238.629} C_VEL
LIN {X 0,Y 152.937,Z 444.101,A -85,B 0,C 180,E1 -24240.27,E2 -24240.27} C_VEL
LIN {X 0,Y 154.029,Z 431.574,A -85,B 0,C 180,E1 -24241.363,E2 -24241.363} C_VEL
LIN {X 0,Y 156.762,Z 390.207,A -85,B 0,C 180,E1 -24243.947,E2 -24243.947} C_VEL
LIN {X 0,Y 154.171,Z 358.4,A -85,B 0,C 180,E1 -24246.475,E2 -24246.475} C_VEL
LIN {X 0,Y 146.416,Z 333.406,A -85,B 0,C 180,E1 -24249.419,E2 -24249.419} C_VEL
LIN {X 0,Y 143.795,Z 325.53,A -85,B 0,C 180,E1 -24250.455,E2 -24250.455} C_VEL
LIN {X 0,Y 143.158,Z 322.653,A -85,B 0,C 180,E1 -24252.313,E2 -24252.313} C_VEL
LIN {X 0,Y 143.038,Z 322.664,A -85,B 0,C 180,E1 -24257.478,E2 -24257.478} C_VEL
LIN {X 0,Y 143.072,Z 322.661,A -85,B 0,C 180,E1 -24261.809,E2 -24261.809} C_VEL
LIN {X 0,Y 143.168,Z 322.652,A -85,B 0,C 180,E1 -24267.316,E2 -24267.316} C_VEL
LIN {X 0,Y 143.173,Z 322.65,A -85,B 0,C 180,E1 -24272.076,E2 -24272.076} C_VEL
LIN {X 0,Y 143.219,Z 322.641,A -85,B 0,C 180,E1 -24278.803,E2 -24278.803} C_VEL
LIN {X 0,Y 143.25,Z 322.641,A -85,B 0,C 180,E1 -24282.879,E2 -24282.879} C_VEL
LIN {X 0,Y 143.527,Z 322.605,A -85,B 0,C 180,E1 -24288.703,E2 -24288.703} C_VEL
LIN {X 0,Y 143.601,Z 322.595,A -85,B 0,C 180,E1 -24291.556,E2 -24291.556} C_VEL
LIN {X 0,Y 144.161,Z 322.525,A -85,B 0,C 180,E1 -24299.999,E2 -24299.999} C_VEL
LIN {X 0,Y 143.6,Z 322.595,A -85,B 0,C 180,E1 -24308.442,E2 -24308.442} C_VEL
LIN {X 0,Y 143.492,Z 322.606,A -85,B 0,C 180,E1 -24311.608,E2 -24311.608} C_VEL
LIN {X 0,Y 143.248,Z 322.64,A -85,B 0,C 180,E1 -24317.118,E2 -24317.118} C_VEL
LIN {X 0,Y 143.22,Z 322.642,A -85,B 0,C 180,E1 -24321.198,E2 -24321.198} C_VEL
LIN {X 0,Y 143.184,Z 322.644,A -85,B 0,C 180,E1 -24327.933,E2 -24327.933} C_VEL
LIN {X 0,Y 143.139,Z 322.654,A -85,B 0,C 180,E1 -24333.417,E2 -24333.417} C_VEL
LIN {X 0,Y 143.058,Z 322.665,A -85,B 0,C 180,E1 -24339.689,E2 -24339.689} C_VEL
LIN {X 0,Y 143.059,Z 322.661,A -85,B 0,C 180,E1 -24343.452,E2 -24343.452} C_VEL
LIN {X 0,Y 143.087,Z 322.66,A -85,B 0,C 180,E1 -24347.454,E2 -24347.454} C_VEL
LIN {X 0,Y 143.124,Z 322.653,A -85,B 0,C 180,E1 -24351.78,E2 -24351.78} C_VEL
LIN {X 0,Y 143.183,Z 322.648,A -85,B 0,C 180,E1 -24357.32,E2 -24357.32} C_VEL
LIN {X 0,Y 143.187,Z 322.644,A -85,B 0,C 180,E1 -24362.063,E2 -24362.063} C_VEL
LIN {X 0,Y 143.276,Z 322.632,A -85,B 0,C 180,E1 -24368.744,E2 -24368.744} C_VEL
LIN {X 0,Y 143.301,Z 322.634,A -85,B 0,C 180,E1 -24372.884,E2 -24372.884} C_VEL
LIN {X 0,Y 143.593,Z 322.594,A -85,B 0,C 180,E1 -24378.707,E2 -24378.707} C_VEL
LIN {X 0,Y 143.674,Z 322.587,A -85,B 0,C 180,E1 -24381.558,E2 -24381.558} C_VEL
LIN {X 0,Y 144.175,Z 322.525,A -85,B 0,C 180,E1 -24389.996,E2 -24389.996} C_VEL
LIN {X 0,Y 143.678,Z 322.589,A -85,B 0,C 180,E1 -24398.433,E2 -24398.433} C_VEL
LIN {X 0,Y 143.566,Z 322.6,A -85,B 0,C 180,E1 -24401.752,E2 -24401.752} C_VEL
LIN {X 0,Y 143.329,Z 322.626,A -85,B 0,C 180,E1 -24407.103,E2 -24407.103} C_VEL
LIN {X 0,Y 143.273,Z 322.636,A -85,B 0,C 180,E1 -24411.925,E2 -24411.925} C_VEL
LIN {X 0,Y 143.252,Z 322.639,A -85,B 0,C 180,E1 -24412.587,E2 -24412.587} C_VEL
LIN {X 0,Y 145.271,Z 328.032,A -85,B 0,C 180,E1 -24413.345,E2 -24413.345} C_VEL
LIN {X 0,Y 153.574,Z 349.044,A -85,B 0,C 180,E1 -24416.093,E2 -24416.093} C_VEL
LIN {X 0,Y 157.937,Z 360.912,A -85,B 0,C 180,E1 -24417.499,E2 -24417.499} C_VEL
LIN {X 0,Y 153.949,Z 418.299,A -85,B 0,C 180,E1 -24421.057,E2 -24421.057} C_VEL
LIN {X 0,Y 153.033,Z 429.491,A -85,B 0,C 180,E1 -24422.144,E2 -24422.144} C_VEL
LIN {X 0,Y 151.297,Z 443.559,A -85,B 0,C 180,E1 -24424.028,E2 -24424.028} C_VEL
LIN {X 0,Y 149.363,Z 456.057,A -85,B 0,C 180,E1 -24426.316,E2 -24426.316} C_VEL
LIN {X 0,Y 147.479,Z 467.187,A -85,B 0,C 180,E1 -24428.943,E2 -24428.943} C_VEL
LIN {X 0,Y 145.471,Z 478.057,A -85,B 0,C 180,E1 -24432.181,E2 -24432.181} C_VEL
LIN {X 0,Y 143.748,Z 487.805,A -85,B 0,C 180,E1 -24435.839,E2 -24435.839} C_VEL
LIN {X 0,Y 142.278,Z 496.786,A -85,B 0,C 180,E1 -24440.05,E2 -24440.05} C_VEL
LIN {X 0,Y 141.367,Z 503.901,A -85,B 0,C 180,E1 -24444.259,E2 -24444.259} C_VEL
LIN {X 0,Y 140.693,Z 510.275,A -85,B 0,C 180,E1 -24449.03,E2 -24449.03} C_VEL
LIN {X 0,Y 140.628,Z 515.412,A -85,B 0,C 180,E1 -24454.078,E2 -24454.078} C_VEL
LIN {X 0,Y 141.218,Z 518.45,A -85,B 0,C 180,E1 -24458.085,E2 -24458.085} C_VEL
LIN {X 0,Y 142.698,Z 521.046,A -85,B 0,C 180,E1 -24462.814,E2 -24462.814} C_VEL
LIN {X 0,Y 144.498,Z 522.325,A -85,B 0,C 180,E1 -24466.549,E2 -24466.549} C_VEL
LIN {X 0,Y 148.149,Z 522.968,A -85,B 0,C 180,E1 -24471.819,E2 -24471.819} C_VEL
LIN {X 0,Y 150.678,Z 522.695,A -85,B 0,C 180,E1 -24474.649,E2 -24474.649} C_VEL
LIN {X 0,Y 154.656,Z 521.585,A -85,B 0,C 180,E1 -24478.318,E2 -24478.318} C_VEL
LIN {X 0,Y 160.412,Z 519.047,A -85,B 0,C 180,E1 -24482.512,E2 -24482.512} C_VEL
LIN {X 0,Y 166.358,Z 515.58,A -85,B 0,C 180,E1 -24486.064,E2 -24486.064} C_VEL
LIN {X 0,Y 173.025,Z 510.821,A -85,B 0,C 180,E1 -24489.352,E2 -24489.352} C_VEL
LIN {X 0,Y 180.518,Z 504.467,A -85,B 0,C 180,E1 -24492.481,E2 -24492.481} C_VEL
LIN {X 0,Y 188.076,Z 496.924,A -85,B 0,C 180,E1 -24495.165,E2 -24495.165} C_VEL
LIN {X 0,Y 194.864,Z 488.898,A -85,B 0,C 180,E1 -24497.311,E2 -24497.311} C_VEL
LIN {X 0,Y 202.652,Z 478.122,A -85,B 0,C 180,E1 -24499.489,E2 -24499.489} C_VEL
LIN {X 0,Y 208.582,Z 468.292,A -85,B 0,C 180,E1 -24500.978,E2 -24500.978} C_VEL
LIN {X 0,Y 214.346,Z 456.754,A -85,B 0,C 180,E1 -24502.324,E2 -24502.324} C_VEL
LIN {X 0,Y 219.056,Z 445.02,A -85,B 0,C 180,E1 -24503.373,E2 -24503.373} C_VEL
LIN {X 0,Y 223.309,Z 431.159,A -85,B 0,C 180,E1 -24504.274,E2 -24504.274} C_VEL
LIN {X 0,Y 226.036,Z 418.635,A -85,B 0,C 180,E1 -24504.83,E2 -24504.83} C_VEL
LIN {X 0,Y 226.575,Z 415.43,A -85,B 0,C 180,E1 -24504.978,E2 -24504.978} C_VEL
LIN {X 0,Y 225.611,Z 413.643,A -85,B 0,C 180,E1 -24507.858,E2 -24507.858} C_VEL
LIN {X 0,Y 225.213,Z 413.577,A -85,B 0,C 180,E1 -24510.383,E2 -24510.383} C_VEL
LIN {X 0,Y 225.259,Z 414.193,A -85,B 0,C 180,E1 -24511.915,E2 -24511.915} C_VEL
LIN {X 0,Y 225.6,Z 417.555,A -85,B 0,C 180,E1 -24514.961,E2 -24514.961} C_VEL
LIN {X 0,Y 225.929,Z 420.067,A -85,B 0,C 180,E1 -24516.407,E2 -24516.407} C_VEL
LIN {X 0,Y 222.926,Z 434.402,A -85,B 0,C 180,E1 -24516.975,E2 -24516.975} C_VEL
LIN {X 0,Y 218.675,Z 448.418,A -85,B 0,C 180,E1 -24517.695,E2 -24517.695} C_VEL
LIN {X 0,Y 213.487,Z 461.287,A -85,B 0,C 180,E1 -24518.582,E2 -24518.582} C_VEL
LIN {X 0,Y 207.644,Z 472.91,A -85,B 0,C 180,E1 -24519.658,E2 -24519.658} C_VEL
LIN {X 0,Y 200.602,Z 484.555,A -85,B 0,C 180,E1 -24521.14,E2 -24521.14} C_VEL
LIN {X 0,Y 192.51,Z 495.803,A -85,B 0,C 180,E1 -24523.113,E2 -24523.113} C_VEL
LIN {X 0,Y 184.89,Z 504.941,A -85,B 0,C 180,E1 -24525.325,E2 -24525.325} C_VEL
LIN {X 0,Y 176.515,Z 513.523,A -85,B 0,C 180,E1 -24528.181,E2 -24528.181} C_VEL
LIN {X 0,Y 168.77,Z 520.447,A -85,B 0,C 180,E1 -24531.354,E2 -24531.354} C_VEL
LIN {X 0,Y 162.891,Z 525.136,A -85,B 0,C 180,E1 -24534.385,E2 -24534.385} C_VEL
LIN {X 0,Y 157.45,Z 528.85,A -85,B 0,C 180,E1 -24537.621,E2 -24537.621} C_VEL
LIN {X 0,Y 151.468,Z 532.476,A -85,B 0,C 180,E1 -24542.363,E2 -24542.363} C_VEL
LIN {X 0,Y 146.654,Z 534.585,A -85,B 0,C 180,E1 -24547.464,E2 -24547.464} C_VEL
LIN {X 0,Y 143.211,Z 535.292,A -85,B 0,C 180,E1 -24552.882,E2 -24552.882} C_VEL
LIN {X 0,Y 141.497,Z 534.593,A -85,B 0,C 180,E1 -24558.546,E2 -24558.546} C_VEL
LIN {X 0,Y 141.275,Z 534.065,A -85,B 0,C 180,E1 -24560.211,E2 -24560.211} C_VEL
LIN {X 0,Y 140.484,Z 533.124,A -85,B 0,C 180,E1 -24562.558,E2 -24562.558} C_VEL
LIN {X 0,Y 138.943,Z 531.737,A -85,B 0,C 180,E1 -24564.845,E2 -24564.845} C_VEL
LIN {X 0,Y 135.522,Z 527.939,A -85,B 0,C 180,E1 -24569.401,E2 -24569.401} C_VEL
LIN {X 0,Y 134.552,Z 524.8,A -85,B 0,C 180,E1 -24572.52,E2 -24572.52} C_VEL
LIN {X 0,Y 134.597,Z 519.198,A -85,B 0,C 180,E1 -24577.201,E2 -24577.201} C_VEL
LIN {X 0,Y 135.117,Z 511.763,A -85,B 0,C 180,E1 -24582.012,E2 -24582.012} C_VEL
LIN {X 0,Y 136.309,Z 502.912,A -85,B 0,C 180,E1 -24586.477,E2 -24586.477} C_VEL
LIN {X 0,Y 137.802,Z 493.825,A -85,B 0,C 180,E1 -24590.139,E2 -24590.139} C_VEL
LIN {X 0,Y 139.684,Z 483.876,A -85,B 0,C 180,E1 -24593.345,E2 -24593.345} C_VEL
LIN {X 0,Y 141.939,Z 471.462,A -85,B 0,C 180,E1 -24596.466,E2 -24596.466} C_VEL
LIN {X 0,Y 144.043,Z 458.68,A -85,B 0,C 180,E1 -24598.886,E2 -24598.886} C_VEL
LIN {X 0,Y 145.941,Z 445.005,A -85,B 0,C 180,E1 -24600.776,E2 -24600.776} C_VEL
LIN {X 0,Y 147.046,Z 433.098,A -85,B 0,C 180,E1 -24601.921,E2 -24601.921} C_VEL
LIN {X 0,Y 149.928,Z 390.355,A -85,B 0,C 180,E1 -24604.733,E2 -24604.733} C_VEL
LIN {X 0,Y 147.539,Z 360.176,A -85,B 0,C 180,E1 -24607.264,E2 -24607.264} C_VEL
LIN {X 0,Y 140.328,Z 336.623,A -85,B 0,C 180,E1 -24610.132,E2 -24610.132} C_VEL
LIN {X 0,Y 136.434,Z 325.065,A -85,B 0,C 180,E1 -24611.785,E2 -24611.785} C_VEL
LIN {X 0,Y 136.108,Z 323.532,A -85,B 0,C 180,E1 -24612.846,E2 -24612.846} C_VEL
LIN {X 0,Y 135.982,Z 323.544,A -85,B 0,C 180,E1 -24617.786,E2 -24617.786} C_VEL
LIN {X 0,Y 136.02,Z 323.54,A -85,B 0,C 180,E1 -24621.68,E2 -24621.68} C_VEL
LIN {X 0,Y 136.05,Z 323.537,A -85,B 0,C 180,E1 -24625.743,E2 -24625.743} C_VEL
LIN {X 0,Y 136.114,Z 323.529,A -85,B 0,C 180,E1 -24632.308,E2 -24632.308} C_VEL
LIN {X 0,Y 136.183,Z 323.518,A -85,B 0,C 180,E1 -24638.821,E2 -24638.821} C_VEL
LIN {X 0,Y 136.221,Z 323.512,A -85,B 0,C 180,E1 -24645.049,E2 -24645.049} C_VEL
LIN {X 0,Y 136.424,Z 323.49,A -85,B 0,C 180,E1 -24648.177,E2 -24648.177} C_VEL
LIN {X 0,Y 136.531,Z 323.478,A -85,B 0,C 180,E1 -24651.115,E2 -24651.115} C_VEL
LIN {X 0,Y 137.119,Z 323.402,A -85,B 0,C 180,E1 -24659.999,E2 -24659.999} C_VEL
LIN {X 0,Y 136.529,Z 323.476,A -85,B 0,C 180,E1 -24668.882,E2 -24668.882} C_VEL
LIN {X 0,Y 136.41,Z 323.49,A -85,B 0,C 180,E1 -24671.891,E2 -24671.891} C_VEL
LIN {X 0,Y 136.16,Z 323.519,A -85,B 0,C 180,E1 -24678.039,E2 -24678.039} C_VEL
LIN {X 0,Y 136.147,Z 323.525,A -85,B 0,C 180,E1 -24681.696,E2 -24681.696} C_VEL
LIN {X 0,Y 136.094,Z 323.529,A -85,B 0,C 180,E1 -24688.612,E2 -24688.612} C_VEL
LIN {X 0,Y 136.039,Z 323.535,A -85,B 0,C 180,E1 -24694.628,E2 -24694.628} C_VEL
LIN {X 0,Y 136.028,Z 323.539,A -85,B 0,C 180,E1 -24699.196,E2 -24699.196} C_VEL
LIN {X 0,Y 136.001,Z 323.54,A -85,B 0,C 180,E1 -24703.658,E2 -24703.658} C_VEL
LIN {X 0,Y 136.049,Z 323.538,A -85,B 0,C 180,E1 -24707.812,E2 -24707.812} C_VEL
LIN {X 0,Y 136.074,Z 323.532,A -85,B 0,C 180,E1 -24711.698,E2 -24711.698} C_VEL
LIN {X 0,Y 136.09,Z 323.532,A -85,B 0,C 180,E1 -24715.715,E2 -24715.715} C_VEL
LIN {X 0,Y 136.143,Z 323.522,A -85,B 0,C 180,E1 -24722.313,E2 -24722.313} C_VEL
LIN {X 0,Y 136.243,Z 323.508,A -85,B 0,C 180,E1 -24728.83,E2 -24728.83} C_VEL
LIN {X 0,Y 136.272,Z 323.509,A -85,B 0,C 180,E1 -24735.053,E2 -24735.053} C_VEL
LIN {X 0,Y 136.496,Z 323.476,A -85,B 0,C 180,E1 -24738.111,E2 -24738.111} C_VEL
LIN {X 0,Y 136.598,Z 323.469,A -85,B 0,C 180,E1 -24741.117,E2 -24741.117} C_VEL
LIN {X 0,Y 137.132,Z 323.402,A -85,B 0,C 180,E1 -24749.995,E2 -24749.995} C_VEL
LIN {X 0,Y 136.602,Z 323.47,A -85,B 0,C 180,E1 -24758.873,E2 -24758.873} C_VEL
LIN {X 0,Y 136.488,Z 323.481,A -85,B 0,C 180,E1 -24761.954,E2 -24761.954} C_VEL
LIN {X 0,Y 136.267,Z 323.509,A -85,B 0,C 180,E1 -24768.019,E2 -24768.019} C_VEL
LIN {X 0,Y 136.255,Z 323.519,A -85,B 0,C 180,E1 -24771.451,E2 -24771.451} C_VEL
LIN {X 0,Y 138.639,Z 329.93,A -85,B 0,C 180,E1 -24772.394,E2 -24772.394} C_VEL
LIN {X 0,Y 146.362,Z 349.41,A -85,B 0,C 180,E1 -24775.121,E2 -24775.121} C_VEL
LIN {X 0,Y 151.178,Z 362.963,A -85,B 0,C 180,E1 -24776.762,E2 -24776.762} C_VEL
LIN {X 0,Y 147.048,Z 418.881,A -85,B 0,C 180,E1 -24780.412,E2 -24780.412} C_VEL
LIN {X 0,Y 146.098,Z 429.765,A -85,B 0,C 180,E1 -24781.521,E2 -24781.521} C_VEL
LIN {X 0,Y 144.367,Z 443.498,A -85,B 0,C 180,E1 -24783.448,E2 -24783.448} C_VEL
LIN {X 0,Y 142.412,Z 455.795,A -85,B 0,C 180,E1 -24785.779,E2 -24785.779} C_VEL
LIN {X 0,Y 140.442,Z 467.183,A -85,B 0,C 180,E1 -24788.567,E2 -24788.567} C_VEL
LIN {X 0,Y 138.454,Z 477.641,A -85,B 0,C 180,E1 -24791.782,E2 -24791.782} C_VEL
LIN {X 0,Y 136.805,Z 486.748,A -85,B 0,C 180,E1 -24795.281,E2 -24795.281} C_VEL
LIN {X 0,Y 135.315,Z 495.643,A -85,B 0,C 180,E1 -24799.519,E2 -24799.519} C_VEL
LIN {X 0,Y 134.332,Z 503.143,A -85,B 0,C 180,E1 -24803.981,E2 -24803.981} C_VEL
LIN {X 0,Y 133.693,Z 508.895,A -85,B 0,C 180,E1 -24808.288,E2 -24808.288} C_VEL
LIN {X 0,Y 133.537,Z 514.302,A -85,B 0,C 180,E1 -24813.448,E2 -24813.448} C_VEL
LIN {X 0,Y 134.214,Z 518.292,A -85,B 0,C 180,E1 -24818.499,E2 -24818.499} C_VEL
LIN {X 0,Y 135.154,Z 520.295,A -85,B 0,C 180,E1 -24821.822,E2 -24821.822} C_VEL
LIN {X 0,Y 137.265,Z 522.303,A -85,B 0,C 180,E1 -24826.562,E2 -24826.562} C_VEL
LIN {X 0,Y 141.61,Z 523.447,A -85,B 0,C 180,E1 -24832.935,E2 -24832.935} C_VEL
LIN {X 0,Y 147.592,Z 522.675,A -85,B 0,C 180,E1 -24838.844,E2 -24838.844} C_VEL
LIN {X 0,Y 152.641,Z 521,A -85,B 0,C 180,E1 -24842.64,E2 -24842.64} C_VEL
LIN {X 0,Y 158.642,Z 518.172,A -85,B 0,C 180,E1 -24846.36,E2 -24846.36} C_VEL
LIN {X 0,Y 165.442,Z 514.121,A -85,B 0,C 180,E1 -24849.784,E2 -24849.784} C_VEL
LIN {X 0,Y 173.11,Z 508.565,A -85,B 0,C 180,E1 -24853.044,E2 -24853.044} C_VEL
LIN {X 0,Y 180.723,Z 501.978,A -85,B 0,C 180,E1 -24855.797,E2 -24855.797} C_VEL
LIN {X 0,Y 189.152,Z 493.351,A -85,B 0,C 180,E1 -24858.411,E2 -24858.411} C_VEL
LIN {X 0,Y 196.731,Z 484.117,A -85,B 0,C 180,E1 -24860.488,E2 -24860.488} C_VEL
LIN {X 0,Y 203.221,Z 474.749,A -85,B 0,C 180,E1 -24862.093,E2 -24862.093} C_VEL
LIN {X 0,Y 210.24,Z 462.557,A -85,B 0,C 180,E1 -24863.651,E2 -24863.651} C_VEL
LIN {X 0,Y 214.939,Z 452.632,A -85,B 0,C 180,E1 -24864.64,E2 -24864.64} C_VEL
LIN {X 0,Y 219.464,Z 440.806,A -85,B 0,C 180,E1 -24865.543,E2 -24865.543} C_VEL
LIN {X 0,Y 223.167,Z 427.758,A -85,B 0,C 180,E1 -24866.264,E2 -24866.264} C_VEL
LIN {X 0,Y 224.551,Z 421.342,A -85,B 0,C 180,E1 -24866.531,E2 -24866.531} C_VEL
LIN {X 0,Y 224.108,Z 420.484,A -85,B 0,C 180,E1 -24868.605,E2 -24868.605} C_VEL
LIN {X 0,Y 223.884,Z 420.86,A -85,B 0,C 180,E1 -24871.379,E2 -24871.379} C_VEL
LIN {X 0,Y 224.004,Z 424.205,A -85,B 0,C 180,E1 -24874.453,E2 -24874.453} C_VEL
LIN {X 0,Y 224.016,Z 424.955,A -85,B 0,C 180,E1 -24874.805,E2 -24874.805} C_VEL
LIN {X 0,Y 220.675,Z 438.474,A -85,B 0,C 180,E1 -24875.338,E2 -24875.338} C_VEL
LIN {X 0,Y 216.542,Z 450.509,A -85,B 0,C 180,E1 -24875.964,E2 -24875.964} C_VEL
LIN {X 0,Y 210.799,Z 463.559,A -85,B 0,C 180,E1 -24876.868,E2 -24876.868} C_VEL
LIN {X 0,Y 204.085,Z 475.786,A -85,B 0,C 180,E1 -24878.038,E2 -24878.038} C_VEL
LIN {X 0,Y 196.87,Z 486.814,A -85,B 0,C 180,E1 -24879.48,E2 -24879.48} C_VEL
LIN {X 0,Y 189.227,Z 496.685,A -85,B 0,C 180,E1 -24881.24,E2 -24881.24} C_VEL
LIN {X 0,Y 181.304,Z 505.457,A -85,B 0,C 180,E1 -24883.391,E2 -24883.391} C_VEL
LIN {X 0,Y 173.786,Z 512.78,A -85,B 0,C 180,E1 -24885.776,E2 -24885.776} C_VEL
LIN {X 0,Y 165.591,Z 519.697,A -85,B 0,C 180,E1 -24888.874,E2 -24888.874} C_VEL
LIN {X 0,Y 157.193,Z 525.753,A -85,B 0,C 180,E1 -24892.883,E2 -24892.883} C_VEL
LIN {X 0,Y 151.524,Z 529.233,A -85,B 0,C 180,E1 -24896.189,E2 -24896.189} C_VEL
LIN {X 0,Y 145.193,Z 532.488,A -85,B 0,C 180,E1 -24901.058,E2 -24901.058} C_VEL
LIN {X 0,Y 140.097,Z 534.353,A -85,B 0,C 180,E1 -24906.347,E2 -24906.347} C_VEL
LIN {X 0,Y 136.427,Z 534.764,A -85,B 0,C 180,E1 -24912.003,E2 -24912.003} C_VEL
LIN {X 0,Y 134.567,Z 533.785,A -85,B 0,C 180,E1 -24917.948,E2 -24917.948} C_VEL
LIN {X 0,Y 134.158,Z 531.365,A -85,B 0,C 180,E1 -24923.991,E2 -24923.991} C_VEL
LIN {X 0,Y 134.449,Z 528.44,A -85,B 0,C 180,E1 -24928.507,E2 -24928.507} C_VEL
LIN {X 0,Y 134.554,Z 525.855,A -85,B 0,C 180,E1 -24931.501,E2 -24931.501} C_VEL
LIN {X 0,Y 134.552,Z 524.8,A -85,B 0,C 180,E1 -24932.52,E2 -24932.52} C_VEL
LIN {X 0,Y 133.929,Z 522.21,A -85,B 0,C 180,E1 -24934.762,E2 -24934.762} C_VEL
LIN {X 0,Y 132.414,Z 519.261,A -85,B 0,C 180,E1 -24936.891,E2 -24936.891} C_VEL
LIN {X 0,Y 128.689,Z 511.39,A -85,B 0,C 180,E1 -24941.716,E2 -24941.716} C_VEL
LIN {X 0,Y 128.44,Z 507.626,A -85,B 0,C 180,E1 -24943.783,E2 -24943.783} C_VEL
LIN {X 0,Y 129.83,Z 498.592,A -85,B 0,C 180,E1 -24948.139,E2 -24948.139} C_VEL
LIN {X 0,Y 131.638,Z 488.668,A -85,B 0,C 180,E1 -24951.948,E2 -24951.948} C_VEL
LIN {X 0,Y 133.752,Z 477.575,A -85,B 0,C 180,E1 -24955.275,E2 -24955.275} C_VEL
LIN {X 0,Y 135.821,Z 465.858,A -85,B 0,C 180,E1 -24958.018,E2 -24958.018} C_VEL
LIN {X 0,Y 137.629,Z 454.875,A -85,B 0,C 180,E1 -24959.992,E2 -24959.992} C_VEL
LIN {X 0,Y 139.493,Z 440.776,A -85,B 0,C 180,E1 -24961.834,E2 -24961.834} C_VEL
LIN {X 0,Y 140.625,Z 427.155,A -85,B 0,C 180,E1 -24963.03,E2 -24963.03} C_VEL
LIN {X 0,Y 143.153,Z 391.034,A -85,B 0,C 180,E1 -24965.505,E2 -24965.505} C_VEL
LIN {X 0,Y 140.868,Z 361.784,A -85,B 0,C 180,E1 -24968.061,E2 -24968.061} C_VEL
LIN {X 0,Y 134.181,Z 339.592,A -85,B 0,C 180,E1 -24970.932,E2 -24970.932} C_VEL
LIN {X 0,Y 129.073,Z 324.587,A -85,B 0,C 180,E1 -24973.257,E2 -24973.257} C_VEL
LIN {X 0,Y 128.935,Z 324.425,A -85,B 0,C 180,E1 -24979.74,E2 -24979.74} C_VEL
LIN {X 0,Y 128.955,Z 324.422,A -85,B 0,C 180,E1 -24984.835,E2 -24984.835} C_VEL
LIN {X 0,Y 129.018,Z 324.413,A -85,B 0,C 180,E1 -24990.641,E2 -24990.641} C_VEL
LIN {X 0,Y 129.068,Z 324.403,A -85,B 0,C 180,E1 -24997.77,E2 -24997.77} C_VEL
LIN {X 0,Y 129.143,Z 324.394,A -85,B 0,C 180,E1 -25004.209,E2 -25004.209} C_VEL
LIN {X 0,Y 129.341,Z 324.372,A -85,B 0,C 180,E1 -25007.973,E2 -25007.973} C_VEL
LIN {X 0,Y 129.457,Z 324.358,A -85,B 0,C 180,E1 -25010.625,E2 -25010.625} C_VEL
LIN {X 0,Y 130.075,Z 324.28,A -85,B 0,C 180,E1 -25019.998,E2 -25019.998} C_VEL
LIN {X 0,Y 129.456,Z 324.356,A -85,B 0,C 180,E1 -25029.372,E2 -25029.372} C_VEL
LIN {X 0,Y 129.294,Z 324.377,A -85,B 0,C 180,E1 -25032.556,E2 -25032.556} C_VEL
LIN {X 0,Y 129.079,Z 324.4,A -85,B 0,C 180,E1 -25039.066,E2 -25039.066} C_VEL
LIN {X 0,Y 129.045,Z 324.41,A -85,B 0,C 180,E1 -25042.408,E2 -25042.408} C_VEL
LIN {X 0,Y 129.011,Z 324.411,A -85,B 0,C 180,E1 -25045.835,E2 -25045.835} C_VEL
LIN {X 0,Y 129.015,Z 324.411,A -85,B 0,C 180,E1 -25049.356,E2 -25049.356} C_VEL
LIN {X 0,Y 128.956,Z 324.417,A -85,B 0,C 180,E1 -25055.165,E2 -25055.165} C_VEL
LIN {X 0,Y 128.932,Z 324.424,A -85,B 0,C 180,E1 -25060.85,E2 -25060.85} C_VEL
LIN {X 0,Y 128.926,Z 324.42,A -85,B 0,C 180,E1 -25065.123,E2 -25065.123} C_VEL
LIN {X 0,Y 128.992,Z 324.417,A -85,B 0,C 180,E1 -25069.707,E2 -25069.707} C_VEL
LIN {X 0,Y 128.996,Z 324.415,A -85,B 0,C 180,E1 -25074.806,E2 -25074.806} C_VEL
LIN {X 0,Y 129.016,Z 324.407,A -85,B 0,C 180,E1 -25080.64,E2 -25080.64} C_VEL
LIN {X 0,Y 129.027,Z 324.412,A -85,B 0,C 180,E1 -25084.164,E2 -25084.164} C_VEL
LIN {X 0,Y 129.107,Z 324.401,A -85,B 0,C 180,E1 -25087.725,E2 -25087.725} C_VEL
LIN {X 0,Y 129.153,Z 324.395,A -85,B 0,C 180,E1 -25090.94,E2 -25090.94} C_VEL
LIN {X 0,Y 129.416,Z 324.358,A -85,B 0,C 180,E1 -25097.815,E2 -25097.815} C_VEL
LIN {X 0,Y 129.522,Z 324.351,A -85,B 0,C 180,E1 -25100.627,E2 -25100.627} C_VEL
LIN {X 0,Y 130.087,Z 324.28,A -85,B 0,C 180,E1 -25109.995,E2 -25109.995} C_VEL
LIN {X 0,Y 129.525,Z 324.35,A -85,B 0,C 180,E1 -25119.362,E2 -25119.362} C_VEL
LIN {X 0,Y 129.39,Z 324.367,A -85,B 0,C 180,E1 -25122.542,E2 -25122.542} C_VEL
LIN {X 0,Y 129.191,Z 324.395,A -85,B 0,C 180,E1 -25130.181,E2 -25130.181} C_VEL
LIN {X 0,Y 131.926,Z 331.477,A -85,B 0,C 180,E1 -25131.323,E2 -25131.323} C_VEL
LIN {X 0,Y 139.761,Z 351.226,A -85,B 0,C 180,E1 -25134.273,E2 -25134.273} C_VEL
LIN {X 0,Y 144.283,Z 363.752,A -85,B 0,C 180,E1 -25135.91,E2 -25135.91} C_VEL
LIN {X 0,Y 140.425,Z 416.031,A -85,B 0,C 180,E1 -25139.45,E2 -25139.45} C_VEL
LIN {X 0,Y 139.436,Z 427.985,A -85,B 0,C 180,E1 -25140.621,E2 -25140.621} C_VEL
LIN {X 0,Y 137.814,Z 440.723,A -85,B 0,C 180,E1 -25142.371,E2 -25142.371} C_VEL
LIN {X 0,Y 135.889,Z 453.108,A -85,B 0,C 180,E1 -25144.664,E2 -25144.664} C_VEL
LIN {X 0,Y 133.854,Z 464.636,A -85,B 0,C 180,E1 -25147.428,E2 -25147.428} C_VEL
LIN {X 0,Y 131.583,Z 476.579,A -85,B 0,C 180,E1 -25151.136,E2 -25151.136} C_VEL
LIN {X 0,Y 129.889,Z 485.648,A -85,B 0,C 180,E1 -25154.688,E2 -25154.688} C_VEL
LIN {X 0,Y 128.363,Z 494.38,A -85,B 0,C 180,E1 -25158.93,E2 -25158.93} C_VEL
LIN {X 0,Y 127.307,Z 502.079,A -85,B 0,C 180,E1 -25163.601,E2 -25163.601} C_VEL
LIN {X 0,Y 126.649,Z 508.159,A -85,B 0,C 180,E1 -25168.187,E2 -25168.187} C_VEL
LIN {X 0,Y 126.462,Z 513.832,A -85,B 0,C 180,E1 -25173.605,E2 -25173.605} C_VEL
LIN {X 0,Y 127.373,Z 518.561,A -85,B 0,C 180,E1 -25179.689,E2 -25179.689} C_VEL
LIN {X 0,Y 128.865,Z 521.101,A -85,B 0,C 180,E1 -25184.177,E2 -25184.177} C_VEL
LIN {X 0,Y 130.523,Z 522.481,A -85,B 0,C 180,E1 -25187.564,E2 -25187.564} C_VEL
LIN {X 0,Y 134.43,Z 523.814,A -85,B 0,C 180,E1 -25193.284,E2 -25193.284} C_VEL
LIN {X 0,Y 137.918,Z 523.912,A -85,B 0,C 180,E1 -25197.081,E2 -25197.081} C_VEL
LIN {X 0,Y 141.176,Z 523.477,A -85,B 0,C 180,E1 -25200.001,E2 -25200.001} C_VEL
LIN {X 0,Y 144.828,Z 522.608,A -85,B 0,C 180,E1 -25202.783,E2 -25202.783} C_VEL
LIN {X 0,Y 148.829,Z 521.231,A -85,B 0,C 180,E1 -25205.421,E2 -25205.421} C_VEL
LIN {X 0,Y 156.914,Z 517.523,A -85,B 0,C 180,E1 -25209.876,E2 -25209.876} C_VEL
LIN {X 0,Y 164.974,Z 512.718,A -85,B 0,C 180,E1 -25213.419,E2 -25213.419} C_VEL
LIN {X 0,Y 173.381,Z 506.541,A -85,B 0,C 180,E1 -25216.485,E2 -25216.485} C_VEL
LIN {X 0,Y 181.955,Z 499.027,A -85,B 0,C 180,E1 -25219.167,E2 -25219.167} C_VEL
LIN {X 0,Y 190.075,Z 490.476,A -85,B 0,C 180,E1 -25221.376,E2 -25221.376} C_VEL
LIN {X 0,Y 198.268,Z 480.242,A -85,B 0,C 180,E1 -25223.333,E2 -25223.333} C_VEL
LIN {X 0,Y 205.129,Z 469.95,A -85,B 0,C 180,E1 -25224.817,E2 -25224.817} C_VEL
LIN {X 0,Y 211.085,Z 459.07,A -85,B 0,C 180,E1 -25225.998,E2 -25225.998} C_VEL
LIN {X 0,Y 216.529,Z 446.759,A -85,B 0,C 180,E1 -25227.028,E2 -25227.028} C_VEL
LIN {X 0,Y 221.025,Z 433.468,A -85,B 0,C 180,E1 -25227.844,E2 -25227.844} C_VEL
LIN {X 0,Y 222.607,Z 427.47,A -85,B 0,C 180,E1 -25228.168,E2 -25228.168} C_VEL
LIN {X 0,Y 222.322,Z 427.666,A -85,B 0,C 180,E1 -25231.022,E2 -25231.022} C_VEL
LIN {X 0,Y 222.18,Z 429.845,A -85,B 0,C 180,E1 -25233.158,E2 -25233.158} C_VEL
LIN {X 0,Y 217.992,Z 443.809,A -85,B 0,C 180,E1 -25233.724,E2 -25233.724} C_VEL
LIN {X 0,Y 212.429,Z 457.645,A -85,B 0,C 180,E1 -25234.527,E2 -25234.527} C_VEL
LIN {X 0,Y 206.791,Z 468.749,A -85,B 0,C 180,E1 -25235.361,E2 -25235.361} C_VEL
LIN {X 0,Y 199.961,Z 479.825,A -85,B 0,C 180,E1 -25236.501,E2 -25236.501} C_VEL
LIN {X 0,Y 193.307,Z 488.985,A -85,B 0,C 180,E1 -25237.757,E2 -25237.757} C_VEL
LIN {X 0,Y 184.765,Z 499.148,A -85,B 0,C 180,E1 -25239.635,E2 -25239.635} C_VEL
LIN {X 0,Y 176.633,Z 507.422,A -85,B 0,C 180,E1 -25241.763,E2 -25241.763} C_VEL
LIN {X 0,Y 167.607,Z 515.226,A -85,B 0,C 180,E1 -25244.545,E2 -25244.545} C_VEL
LIN {X 0,Y 160.377,Z 520.695,A -85,B 0,C 180,E1 -25247.227,E2 -25247.227} C_VEL
LIN {X 0,Y 153.681,Z 525.108,A -85,B 0,C 180,E1 -25250.201,E2 -25250.201} C_VEL
LIN {X 0,Y 145.689,Z 529.546,A -85,B 0,C 180,E1 -25254.638,E2 -25254.638} C_VEL
LIN {X 0,Y 139.005,Z 532.51,A -85,B 0,C 180,E1 -25259.638,E2 -25259.638} C_VEL
LIN {X 0,Y 133.604,Z 534.023,A -85,B 0,C 180,E1 -25265.121,E2 -25265.121} C_VEL
LIN {X 0,Y 129.685,Z 534.165,A -85,B 0,C 180,E1 -25271.032,E2 -25271.032} C_VEL
LIN {X 0,Y 127.627,Z 532.959,A -85,B 0,C 180,E1 -25277.282,E2 -25277.282} C_VEL
LIN {X 0,Y 127.25,Z 531.808,A -85,B 0,C 180,E1 -25280.469,E2 -25280.469} C_VEL
LIN {X 0,Y 127.182,Z 529.996,A -85,B 0,C 180,E1 -25284.096,E2 -25284.096} C_VEL
LIN {X 0,Y 127.49,Z 527.128,A -85,B 0,C 180,E1 -25288.426,E2 -25288.426} C_VEL
LIN {X 0,Y 127.573,Z 524.358,A -85,B 0,C 180,E1 -25291.583,E2 -25291.583} C_VEL
LIN {X 0,Y 127.57,Z 519.072,A -85,B 0,C 180,E1 -25296.33,E2 -25296.33} C_VEL
LIN {X 0,Y 127.913,Z 512.271,A -85,B 0,C 180,E1 -25301.091,E2 -25301.091} C_VEL
LIN {X 0,Y 128.44,Z 507.626,A -85,B 0,C 180,E1 -25303.783,E2 -25303.783} C_VEL
LIN {X 0,Y 128.337,Z 503.765,A -85,B 0,C 180,E1 -25305.74,E2 -25305.74} C_VEL
LIN {X 0,Y 126.617,Z 496.863,A -85,B 0,C 180,E1 -25308.81,E2 -25308.81} C_VEL
LIN {X 0,Y 125.078,Z 489.359,A -85,B 0,C 180,E1 -25311.741,E2 -25311.741} C_VEL
LIN {X 0,Y 125.292,Z 484.584,A -85,B 0,C 180,E1 -25313.413,E2 -25313.413} C_VEL
LIN {X 0,Y 127.39,Z 473.571,A -85,B 0,C 180,E1 -25316.634,E2 -25316.634} C_VEL
LIN {X 0,Y 129.648,Z 460.994,A -85,B 0,C 180,E1 -25319.448,E2 -25319.448} C_VEL
LIN {X 0,Y 131.572,Z 448.617,A -85,B 0,C 180,E1 -25321.511,E2 -25321.511} C_VEL
LIN {X 0,Y 133.141,Z 435.163,A -85,B 0,C 180,E1 -25323.095,E2 -25323.095} C_VEL
LIN {X 0,Y 136.367,Z 391.203,A -85,B 0,C 180,E1 -25326.359,E2 -25326.359} C_VEL
LIN {X 0,Y 134.262,Z 363.492,A -85,B 0,C 180,E1 -25328.927,E2 -25328.927} C_VEL
LIN {X 0,Y 127.927,Z 342.272,A -85,B 0,C 180,E1 -25331.831,E2 -25331.831} C_VEL
LIN {X 0,Y 123.164,Z 328.475,A -85,B 0,C 180,E1 -25334.001,E2 -25334.001} C_VEL
LIN {X 0,Y 122.013,Z 325.869,A -85,B 0,C 180,E1 -25334.487,E2 -25334.487} C_VEL
LIN {X 0,Y 121.926,Z 325.295,A -85,B 0,C 180,E1 -25334.584,E2 -25334.584} C_VEL
LIN {X 0,Y 121.853,Z 325.308,A -85,B 0,C 180,E1 -25340.62,E2 -25340.62} C_VEL
LIN {X 0,Y 121.906,Z 325.3,A -85,B 0,C 180,E1 -25344.793,E2 -25344.793} C_VEL
LIN {X 0,Y 121.927,Z 325.296,A -85,B 0,C 180,E1 -25349.839,E2 -25349.839} C_VEL
LIN {X 0,Y 121.985,Z 325.284,A -85,B 0,C 180,E1 -25357.193,E2 -25357.193} C_VEL
LIN {X 0,Y 122.057,Z 325.279,A -85,B 0,C 180,E1 -25363.266,E2 -25363.266} C_VEL
LIN {X 0,Y 122.285,Z 325.252,A -85,B 0,C 180,E1 -25367.693,E2 -25367.693} C_VEL
LIN {X 0,Y 122.405,Z 325.232,A -85,B 0,C 180,E1 -25373.404,E2 -25373.404} C_VEL
LIN {X 0,Y 123.028,Z 325.157,A -85,B 0,C 180,E1 -25379.998,E2 -25379.998} C_VEL
LIN {X 0,Y 122.373,Z 325.237,A -85,B 0,C 180,E1 -25387.11,E2 -25387.11} C_VEL
LIN {X 0,Y 122.283,Z 325.25,A -85,B 0,C 180,E1 -25392.303,E2 -25392.303} C_VEL
LIN {X 0,Y 122.055,Z 325.279,A -85,B 0,C 180,E1 -25396.731,E2 -25396.731} C_VEL
LIN {X 0,Y 121.987,Z 325.289,A -85,B 0,C 180,E1 -25402.81,E2 -25402.81} C_VEL
LIN {X 0,Y 121.932,Z 325.29,A -85,B 0,C 180,E1 -25407.457,E2 -25407.457} C_VEL
LIN {X 0,Y 121.897,Z 325.3,A -85,B 0,C 180,E1 -25411.256,E2 -25411.256} C_VEL
LIN {X 0,Y 121.881,Z 325.297,A -85,B 0,C 180,E1 -25416.168,E2 -25416.168} C_VEL
LIN {X 0,Y 121.871,Z 325.304,A -85,B 0,C 180,E1 -25421.436,E2 -25421.436} C_VEL
LIN {X 0,Y 121.91,Z 325.299,A -85,B 0,C 180,E1 -25428.539,E2 -25428.539} C_VEL
LIN {X 0,Y 121.949,Z 325.293,A -85,B 0,C 180,E1 -25434.807,E2 -25434.807} C_VEL
LIN {X 0,Y 121.929,Z 325.293,A -85,B 0,C 180,E1 -25439.834,E2 -25439.834} C_VEL
LIN {X 0,Y 121.982,Z 325.291,A -85,B 0,C 180,E1 -25446.212,E2 -25446.212} C_VEL
LIN {X 0,Y 122.044,Z 325.275,A -85,B 0,C 180,E1 -25449.783,E2 -25449.783} C_VEL
LIN {X 0,Y 122.363,Z 325.236,A -85,B 0,C 180,E1 -25457.521,E2 -25457.521} C_VEL
LIN {X 0,Y 122.45,Z 325.229,A -85,B 0,C 180,E1 -25460.081,E2 -25460.081} C_VEL
LIN {X 0,Y 122.607,Z 325.207,A -85,B 0,C 180,E1 -25466.709,E2 -25466.709} C_VEL
LIN {X 0,Y 123.041,Z 325.158,A -85,B 0,C 180,E1 -25469.995,E2 -25469.995} C_VEL
LIN {X 0,Y 122.45,Z 325.231,A -85,B 0,C 180,E1 -25476.586,E2 -25476.586} C_VEL
LIN {X 0,Y 122.452,Z 325.231,A -85,B 0,C 180,E1 -25479.908,E2 -25479.908} C_VEL
LIN {X 0,Y 122.282,Z 325.253,A -85,B 0,C 180,E1 -25483.284,E2 -25483.284} C_VEL
LIN {X 0,Y 122.16,Z 325.43,A -85,B 0,C 180,E1 -25488.874,E2 -25488.874} C_VEL
LIN {X 0,Y 132.174,Z 350.48,A -85,B 0,C 180,E1 -25492.977,E2 -25492.977} C_VEL
LIN {X 0,Y 137.471,Z 365.091,A -85,B 0,C 180,E1 -25495.031,E2 -25495.031} C_VEL
LIN {X 0,Y 134.235,Z 409.007,A -85,B 0,C 180,E1 -25498.125,E2 -25498.125} C_VEL
LIN {X 0,Y 133.118,Z 423.178,A -85,B 0,C 180,E1 -25499.317,E2 -25499.317} C_VEL
LIN {X 0,Y 131.594,Z 435.981,A -85,B 0,C 180,E1 -25500.928,E2 -25500.928} C_VEL
LIN {X 0,Y 129.572,Z 449.245,A -85,B 0,C 180,E1 -25503.253,E2 -25503.253} C_VEL
LIN {X 0,Y 127.491,Z 460.947,A -85,B 0,C 180,E1 -25505.976,E2 -25505.976} C_VEL
LIN {X 0,Y 125.245,Z 472.688,A -85,B 0,C 180,E1 -25509.508,E2 -25509.508} C_VEL
LIN {X 0,Y 123.461,Z 482.127,A -85,B 0,C 180,E1 -25513.074,E2 -25513.074} C_VEL
LIN {X 0,Y 121.646,Z 491.966,A -85,B 0,C 180,E1 -25517.743,E2 -25517.743} C_VEL
LIN {X 0,Y 120.302,Z 501.059,A -85,B 0,C 180,E1 -25523.218,E2 -25523.218} C_VEL
LIN {X 0,Y 119.502,Z 508.484,A -85,B 0,C 180,E1 -25529.032,E2 -25529.032} C_VEL
LIN {X 0,Y 119.413,Z 513.327,A -85,B 0,C 180,E1 -25533.865,E2 -25533.865} C_VEL
LIN {X 0,Y 120.192,Z 517.746,A -85,B 0,C 180,E1 -25539.463,E2 -25539.463} C_VEL
LIN {X 0,Y 121.266,Z 520.063,A -85,B 0,C 180,E1 -25543.157,E2 -25543.157} C_VEL
LIN {X 0,Y 122.84,Z 521.858,A -85,B 0,C 180,E1 -25546.772,E2 -25546.772} C_VEL
LIN {X 0,Y 124.792,Z 523.154,A -85,B 0,C 180,E1 -25550.275,E2 -25550.275} C_VEL
LIN {X 0,Y 127.25,Z 524.031,A -85,B 0,C 180,E1 -25553.692,E2 -25553.692} C_VEL
LIN {X 0,Y 130.064,Z 524.43,A -85,B 0,C 180,E1 -25556.904,E2 -25556.904} C_VEL
LIN {X 0,Y 133.508,Z 524.355,A -85,B 0,C 180,E1 -25560.166,E2 -25560.166} C_VEL
LIN {X 0,Y 136.992,Z 523.883,A -85,B 0,C 180,E1 -25562.942,E2 -25562.942} C_VEL
LIN {X 0,Y 141.28,Z 522.873,A -85,B 0,C 180,E1 -25565.891,E2 -25565.891} C_VEL
LIN {X 0,Y 145.406,Z 521.522,A -85,B 0,C 180,E1 -25568.339,E2 -25568.339} C_VEL
LIN {X 0,Y 152.634,Z 518.438,A -85,B 0,C 180,E1 -25572.017,E2 -25572.017} C_VEL
LIN {X 0,Y 160.39,Z 514.251,A -85,B 0,C 180,E1 -25575.244,E2 -25575.244} C_VEL
LIN {X 0,Y 168.841,Z 508.684,A -85,B 0,C 180,E1 -25578.174,E2 -25578.174} C_VEL
LIN {X 0,Y 176.28,Z 502.795,A -85,B 0,C 180,E1 -25580.418,E2 -25580.418} C_VEL
LIN {X 0,Y 183.982,Z 495.739,A -85,B 0,C 180,E1 -25582.458,E2 -25582.458} C_VEL
LIN {X 0,Y 192.492,Z 486.445,A -85,B 0,C 180,E1 -25584.467,E2 -25584.467} C_VEL
LIN {X 0,Y 200.065,Z 476.53,A -85,B 0,C 180,E1 -25586.048,E2 -25586.048} C_VEL
LIN {X 0,Y 206.843,Z 465.969,A -85,B 0,C 180,E1 -25587.319,E2 -25587.319} C_VEL
LIN {X 0,Y 213.234,Z 453.636,A -85,B 0,C 180,E1 -25588.446,E2 -25588.446} C_VEL
LIN {X 0,Y 217.899,Z 442.268,A -85,B 0,C 180,E1 -25589.226,E2 -25589.226} C_VEL
LIN {X 0,Y 220.482,Z 434.326,A -85,B 0,C 180,E1 -25589.716,E2 -25589.716} C_VEL
LIN {X 0,Y 220.408,Z 434.651,A -85,B 0,C 180,E1 -25591.004,E2 -25591.004} C_VEL
LIN {X 0,Y 220.268,Z 435.375,A -85,B 0,C 180,E1 -25591.512,E2 -25591.512} C_VEL
LIN {X 0,Y 215.621,Z 448.676,A -85,B 0,C 180,E1 -25592.079,E2 -25592.079} C_VEL
LIN {X 0,Y 209.245,Z 462.482,A -85,B 0,C 180,E1 -25592.908,E2 -25592.908} C_VEL
LIN {X 0,Y 202.916,Z 473.428,A -85,B 0,C 180,E1 -25593.788,E2 -25593.788} C_VEL
LIN {X 0,Y 194.448,Z 485.615,A -85,B 0,C 180,E1 -25595.154,E2 -25595.154} C_VEL
LIN {X 0,Y 186.257,Z 495.458,A -85,B 0,C 180,E1 -25596.709,E2 -25596.709} C_VEL
LIN {X 0,Y 177.606,Z 504.228,A -85,B 0,C 180,E1 -25598.613,E2 -25598.613} C_VEL
LIN {X 0,Y 168.03,Z 512.608,A -85,B 0,C 180,E1 -25601.173,E2 -25601.173} C_VEL
LIN {X 0,Y 160.241,Z 518.411,A -85,B 0,C 180,E1 -25603.653,E2 -25603.653} C_VEL
LIN {X 0,Y 152.869,Z 523.125,A -85,B 0,C 180,E1 -25606.412,E2 -25606.412} C_VEL
LIN {X 0,Y 146.182,Z 526.907,A -85,B 0,C 180,E1 -25609.541,E2 -25609.541} C_VEL
LIN {X 0,Y 139.961,Z 529.821,A -85,B 0,C 180,E1 -25612.956,E2 -25612.956} C_VEL
LIN {X 0,Y 132.913,Z 532.425,A -85,B 0,C 180,E1 -25618.087,E2 -25618.087} C_VEL
LIN {X 0,Y 127.181,Z 533.674,A -85,B 0,C 180,E1 -25623.772,E2 -25623.772} C_VEL
LIN {X 0,Y 122.986,Z 533.529,A -85,B 0,C 180,E1 -25629.956,E2 -25629.956} C_VEL
LIN {X 0,Y 120.744,Z 532.005,A -85,B 0,C 180,E1 -25636.543,E2 -25636.543} C_VEL
LIN {X 0,Y 120.184,Z 529.074,A -85,B 0,C 180,E1 -25643.29,E2 -25643.29} C_VEL
LIN {X 0,Y 120.544,Z 525.739,A -85,B 0,C 180,E1 -25648.335,E2 -25648.335} C_VEL
LIN {X 0,Y 120.59,Z 522.83,A -85,B 0,C 180,E1 -25651.675,E2 -25651.675} C_VEL
LIN {X 0,Y 120.608,Z 517.243,A -85,B 0,C 180,E1 -25656.697,E2 -25656.697} C_VEL
LIN {X 0,Y 121.046,Z 510.071,A -85,B 0,C 180,E1 -25661.729,E2 -25661.729} C_VEL
LIN {X 0,Y 122.261,Z 501.13,A -85,B 0,C 180,E1 -25666.707,E2 -25666.707} C_VEL
LIN {X 0,Y 124.038,Z 490.833,A -85,B 0,C 180,E1 -25671.178,E2 -25671.178} C_VEL
LIN {X 0,Y 125.292,Z 484.584,A -85,B 0,C 180,E1 -25673.413,E2 -25673.413} C_VEL
LIN {X 0,Y 125.523,Z 479.759,A -85,B 0,C 180,E1 -25674.972,E2 -25674.972} C_VEL
LIN {X 0,Y 124.185,Z 471.439,A -85,B 0,C 180,E1 -25677.387,E2 -25677.387} C_VEL
LIN {X 0,Y 122.914,Z 462.746,A -85,B 0,C 180,E1 -25679.561,E2 -25679.561} C_VEL
LIN {X 0,Y 123.245,Z 457.333,A -85,B 0,C 180,E1 -25680.679,E2 -25680.679} C_VEL
LIN {X 0,Y 125.31,Z 443.678,A -85,B 0,C 180,E1 -25682.87,E2 -25682.87} C_VEL
LIN {X 0,Y 126.544,Z 431.557,A -85,B 0,C 180,E1 -25684.219,E2 -25684.219} C_VEL
LIN {X 0,Y 129.598,Z 391.607,A -85,B 0,C 180,E1 -25687.284,E2 -25687.284} C_VEL
LIN {X 0,Y 127.649,Z 365.02,A -85,B 0,C 180,E1 -25689.88,E2 -25689.88} C_VEL
LIN {X 0,Y 120.982,Z 342.717,A -85,B 0,C 180,E1 -25693.111,E2 -25693.111} C_VEL
LIN {X 0,Y 117.126,Z 331.752,A -85,B 0,C 180,E1 -25694.993,E2 -25694.993} C_VEL
LIN {X 0,Y 114.987,Z 327.02,A -85,B 0,C 180,E1 -25695.952,E2 -25695.952} C_VEL
LIN {X 0,Y 114.825,Z 326.174,A -85,B 0,C 180,E1 -25696.202,E2 -25696.202} C_VEL
LIN {X 0,Y 114.783,Z 326.184,A -85,B 0,C 180,E1 -25702.749,E2 -25702.749} C_VEL
LIN {X 0,Y 114.855,Z 326.179,A -85,B 0,C 180,E1 -25708.945,E2 -25708.945} C_VEL
LIN {X 0,Y 114.906,Z 326.166,A -85,B 0,C 180,E1 -25716.556,E2 -25716.556} C_VEL
LIN {X 0,Y 114.962,Z 326.164,A -85,B 0,C 180,E1 -25722.2,E2 -25722.2} C_VEL
LIN {X 0,Y 115.302,Z 326.123,A -85,B 0,C 180,E1 -25729.462,E2 -25729.462} C_VEL
LIN {X 0,Y 115.502,Z 326.096,A -85,B 0,C 180,E1 -25736.51,E2 -25736.51} C_VEL
LIN {X 0,Y 115.98,Z 326.035,A -85,B 0,C 180,E1 -25739.998,E2 -25739.998} C_VEL
LIN {X 0,Y 115.345,Z 326.117,A -85,B 0,C 180,E1 -25746.998,E2 -25746.998} C_VEL
LIN {X 0,Y 115.201,Z 326.132,A -85,B 0,C 180,E1 -25752.551,E2 -25752.551} C_VEL
LIN {X 0,Y 114.961,Z 326.16,A -85,B 0,C 180,E1 -25757.797,E2 -25757.797} C_VEL
LIN {X 0,Y 114.914,Z 326.171,A -85,B 0,C 180,E1 -25763.453,E2 -25763.453} C_VEL
LIN {X 0,Y 114.854,Z 326.177,A -85,B 0,C 180,E1 -25771.054,E2 -25771.054} C_VEL
LIN {X 0,Y 114.777,Z 326.184,A -85,B 0,C 180,E1 -25777.755,E2 -25777.755} C_VEL
LIN {X 0,Y 114.788,Z 326.182,A -85,B 0,C 180,E1 -25782.715,E2 -25782.715} C_VEL
LIN {X 0,Y 114.822,Z 326.182,A -85,B 0,C 180,E1 -25787.677,E2 -25787.677} C_VEL
LIN {X 0,Y 114.826,Z 326.175,A -85,B 0,C 180,E1 -25792.716,E2 -25792.716} C_VEL
LIN {X 0,Y 114.863,Z 326.174,A -85,B 0,C 180,E1 -25798.934,E2 -25798.934} C_VEL
LIN {X 0,Y 114.947,Z 326.166,A -85,B 0,C 180,E1 -25806.504,E2 -25806.504} C_VEL
LIN {X 0,Y 115.011,Z 326.157,A -85,B 0,C 180,E1 -25812.206,E2 -25812.206} C_VEL
LIN {X 0,Y 115.284,Z 326.118,A -85,B 0,C 180,E1 -25817.256,E2 -25817.256} C_VEL
LIN {X 0,Y 115.392,Z 326.11,A -85,B 0,C 180,E1 -25822.999,E2 -25822.999} C_VEL
LIN {X 0,Y 115.993,Z 326.036,A -85,B 0,C 180,E1 -25829.994,E2 -25829.994} C_VEL
LIN {X 0,Y 115.392,Z 326.112,A -85,B 0,C 180,E1 -25836.99,E2 -25836.99} C_VEL
LIN {X 0,Y 115.304,Z 326.122,A -85,B 0,C 180,E1 -25842.787,E2 -25842.787} C_VEL
LIN {X 0,Y 115.088,Z 326.143,A -85,B 0,C 180,E1 -25847.312,E2 -25847.312} C_VEL
LIN {X 0,Y 116.061,Z 328.972,A -85,B 0,C 180,E1 -25847.844,E2 -25847.844} C_VEL
LIN {X 0,Y 122.823,Z 345.136,A -85,B 0,C 180,E1 -25850.837,E2 -25850.837} C_VEL
LIN {X 0,Y 130.701,Z 366.424,A -85,B 0,C 180,E1 -25854.092,E2 -25854.092} C_VEL
LIN {X 0,Y 126.956,Z 414.2,A -85,B 0,C 180,E1 -25857.663,E2 -25857.663} C_VEL
LIN {X 0,Y 125.699,Z 427.872,A -85,B 0,C 180,E1 -25859.068,E2 -25859.068} C_VEL
LIN {X 0,Y 124.108,Z 439.939,A -85,B 0,C 180,E1 -25860.843,E2 -25860.843} C_VEL
LIN {X 0,Y 122.023,Z 452.587,A -85,B 0,C 180,E1 -25863.373,E2 -25863.373} C_VEL
LIN {X 0,Y 119.786,Z 464.541,A -85,B 0,C 180,E1 -25866.506,E2 -25866.506} C_VEL
LIN {X 0,Y 117.771,Z 474.663,A -85,B 0,C 180,E1 -25869.884,E2 -25869.884} C_VEL
LIN {X 0,Y 115.663,Z 485.431,A -85,B 0,C 180,E1 -25874.446,E2 -25874.446} C_VEL
LIN {X 0,Y 114.232,Z 493.316,A -85,B 0,C 180,E1 -25878.597,E2 -25878.597} C_VEL
LIN {X 0,Y 113.109,Z 501.374,A -85,B 0,C 180,E1 -25883.86,E2 -25883.86} C_VEL
LIN {X 0,Y 112.46,Z 507.632,A -85,B 0,C 180,E1 -25888.967,E2 -25888.967} C_VEL
LIN {X 0,Y 112.352,Z 512.654,A -85,B 0,C 180,E1 -25894.034,E2 -25894.034} C_VEL
LIN {X 0,Y 113.305,Z 517.683,A -85,B 0,C 180,E1 -25900.461,E2 -25900.461} C_VEL
LIN {X 0,Y 115.518,Z 521.278,A -85,B 0,C 180,E1 -25906.713,E2 -25906.713} C_VEL
LIN {X 0,Y 119.372,Z 523.809,A -85,B 0,C 180,E1 -25913.239,E2 -25913.239} C_VEL
LIN {X 0,Y 122.193,Z 524.619,A -85,B 0,C 180,E1 -25916.704,E2 -25916.704} C_VEL
LIN {X 0,Y 126.497,Z 524.961,A -85,B 0,C 180,E1 -25920.953,E2 -25920.953} C_VEL
LIN {X 0,Y 133.218,Z 524.315,A -85,B 0,C 180,E1 -25926.058,E2 -25926.058} C_VEL
LIN {X 0,Y 137.649,Z 523.293,A -85,B 0,C 180,E1 -25928.812,E2 -25928.812} C_VEL
LIN {X 0,Y 143.687,Z 521.39,A -85,B 0,C 180,E1 -25932.023,E2 -25932.023} C_VEL
LIN {X 0,Y 150.175,Z 518.703,A -85,B 0,C 180,E1 -25934.917,E2 -25934.917} C_VEL
LIN {X 0,Y 158.586,Z 514.354,A -85,B 0,C 180,E1 -25938.074,E2 -25938.074} C_VEL
LIN {X 0,Y 169.059,Z 507.544,A -85,B 0,C 180,E1 -25941.332,E2 -25941.332} C_VEL
LIN {X 0,Y 178.543,Z 499.988,A -85,B 0,C 180,E1 -25943.796,E2 -25943.796} C_VEL
LIN {X 0,Y 187.27,Z 491.541,A -85,B 0,C 180,E1 -25945.771,E2 -25945.771} C_VEL
LIN {X 0,Y 195.933,Z 481.586,A -85,B 0,C 180,E1 -25947.506,E2 -25947.506} C_VEL
LIN {X 0,Y 203.699,Z 470.739,A -85,B 0,C 180,E1 -25948.884,E2 -25948.884} C_VEL
LIN {X 0,Y 210.684,Z 458.625,A -85,B 0,C 180,E1 -25950.026,E2 -25950.026} C_VEL
LIN {X 0,Y 211.191,Z 457.66,A -85,B 0,C 180,E1 -25950.107,E2 -25950.107} C_VEL
LIN {X 0,Y 212.144,Z 455.761,A -85,B 0,C 180,E1 -25950.548,E2 -25950.548} C_VEL
LIN {X 0,Y 205.623,Z 468.015,A -85,B 0,C 180,E1 -25951.313,E2 -25951.313} C_VEL
LIN {X 0,Y 197.866,Z 479.765,A -85,B 0,C 180,E1 -25952.353,E2 -25952.353} C_VEL
LIN {X 0,Y 189.819,Z 489.921,A -85,B 0,C 180,E1 -25953.601,E2 -25953.601} C_VEL
LIN {X 0,Y 180.704,Z 499.612,A -85,B 0,C 180,E1 -25955.255,E2 -25955.255} C_VEL
LIN {X 0,Y 171.936,Z 507.571,A -85,B 0,C 180,E1 -25957.162,E2 -25957.162} C_VEL
LIN {X 0,Y 163.523,Z 514.112,A -85,B 0,C 180,E1 -25959.334,E2 -25959.334} C_VEL
LIN {X 0,Y 155.492,Z 519.533,A -85,B 0,C 180,E1 -25961.787,E2 -25961.787} C_VEL
LIN {X 0,Y 147.845,Z 523.946,A -85,B 0,C 180,E1 -25964.529,E2 -25964.529} C_VEL
LIN {X 0,Y 138.621,Z 528.365,A -85,B 0,C 180,E1 -25968.781,E2 -25968.781} C_VEL
LIN {X 0,Y 130.468,Z 531.367,A -85,B 0,C 180,E1 -25973.673,E2 -25973.673} C_VEL
LIN {X 0,Y 123.768,Z 532.943,A -85,B 0,C 180,E1 -25979.275,E2 -25979.275} C_VEL
LIN {X 0,Y 118.404,Z 533.174,A -85,B 0,C 180,E1 -25985.458,E2 -25985.458} C_VEL
LIN {X 0,Y 114.854,Z 532.081,A -85,B 0,C 180,E1 -25992.192,E2 -25992.192} C_VEL
LIN {X 0,Y 113.367,Z 529.615,A -85,B 0,C 180,E1 -25999.289,E2 -25999.289} C_VEL
LIN {X 0,Y 113.288,Z 526.604,A -85,B 0,C 180,E1 -26004.891,E2 -26004.891} C_VEL
LIN {X 0,Y 113.607,Z 524.285,A -85,B 0,C 180,E1 -26008.233,E2 -26008.233} C_VEL
LIN {X 0,Y 113.633,Z 521.189,A -85,B 0,C 180,E1 -26011.778,E2 -26011.778} C_VEL
LIN {X 0,Y 113.631,Z 515.282,A -85,B 0,C 180,E1 -26017.111,E2 -26017.111} C_VEL
LIN {X 0,Y 114.127,Z 507.771,A -85,B 0,C 180,E1 -26022.451,E2 -26022.451} C_VEL
LIN {X 0,Y 115.573,Z 498.342,A -85,B 0,C 180,E1 -26027.705,E2 -26027.705} C_VEL
LIN {X 0,Y 117.301,Z 488.576,A -85,B 0,C 180,E1 -26031.995,E2 -26031.995} C_VEL
LIN {X 0,Y 119.469,Z 477.791,A -85,B 0,C 180,E1 -26035.715,E2 -26035.715} C_VEL
LIN {X 0,Y 121.727,Z 465.755,A -85,B 0,C 180,E1 -26038.919,E2 -26038.919} C_VEL
LIN {X 0,Y 123.245,Z 457.333,A -85,B 0,C 180,E1 -26040.679,E2 -26040.679} C_VEL
LIN {X 0,Y 123.559,Z 451.876,A -85,B 0,C 180,E1 -26041.698,E2 -26041.698} C_VEL
LIN {X 0,Y 122.82,Z 446.344,A -85,B 0,C 180,E1 -26042.702,E2 -26042.702} C_VEL
LIN {X 0,Y 120.172,Z 433.334,A -85,B 0,C 180,E1 -26044.764,E2 -26044.764} C_VEL
LIN {X 0,Y 120.017,Z 427.539,A -85,B 0,C 180,E1 -26045.386,E2 -26045.386} C_VEL
LIN {X 0,Y 122.819,Z 392.122,A -85,B 0,C 180,E1 -26048.224,E2 -26048.224} C_VEL
LIN {X 0,Y 121.069,Z 366.817,A -85,B 0,C 180,E1 -26050.829,E2 -26050.829} C_VEL
LIN {X 0,Y 114.64,Z 345.033,A -85,B 0,C 180,E1 -26054.231,E2 -26054.231} C_VEL
LIN {X 0,Y 111.161,Z 335.022,A -85,B 0,C 180,E1 -26056.051,E2 -26056.051} C_VEL
LIN {X 0,Y 107.833,Z 327.592,A -85,B 0,C 180,E1 -26057.664,E2 -26057.664} C_VEL
LIN {X 0,Y 107.724,Z 327.063,A -85,B 0,C 180,E1 -26057.908,E2 -26057.908} C_VEL
LIN {X 0,Y 107.711,Z 327.067,A -85,B 0,C 180,E1 -26064.037,E2 -26064.037} C_VEL
LIN {X 0,Y 107.791,Z 327.058,A -85,B 0,C 180,E1 -26068.558,E2 -26068.558} C_VEL
LIN {X 0,Y 107.872,Z 327.041,A -85,B 0,C 180,E1 -26076.987,E2 -26076.987} C_VEL
LIN {X 0,Y 107.967,Z 327.03,A -85,B 0,C 180,E1 -26084.906,E2 -26084.906} C_VEL
LIN {X 0,Y 108.203,Z 327.006,A -85,B 0,C 180,E1 -26088.762,E2 -26088.762} C_VEL
LIN {X 0,Y 108.286,Z 326.993,A -85,B 0,C 180,E1 -26092.54,E2 -26092.54} C_VEL
LIN {X 0,Y 108.906,Z 326.917,A -85,B 0,C 180,E1 -26099.998,E2 -26099.998} C_VEL
LIN {X 0,Y 108.284,Z 326.997,A -85,B 0,C 180,E1 -26107.457,E2 -26107.457} C_VEL
LIN {X 0,Y 108.135,Z 327.013,A -85,B 0,C 180,E1 -26112.865,E2 -26112.865} C_VEL
LIN {X 0,Y 107.859,Z 327.042,A -85,B 0,C 180,E1 -26119.012,E2 -26119.012} C_VEL
LIN {X 0,Y 107.83,Z 327.053,A -85,B 0,C 180,E1 -26124.149,E2 -26124.149} C_VEL
LIN {X 0,Y 107.778,Z 327.06,A -85,B 0,C 180,E1 -26132.035,E2 -26132.035} C_VEL
LIN {X 0,Y 107.687,Z 327.071,A -85,B 0,C 180,E1 -26138.447,E2 -26138.447} C_VEL
LIN {X 0,Y 107.693,Z 327.066,A -85,B 0,C 180,E1 -26145.875,E2 -26145.875} C_VEL
LIN {X 0,Y 107.724,Z 327.062,A -85,B 0,C 180,E1 -26151.523,E2 -26151.523} C_VEL
LIN {X 0,Y 107.803,Z 327.055,A -85,B 0,C 180,E1 -26158.561,E2 -26158.561} C_VEL
LIN {X 0,Y 107.911,Z 327.041,A -85,B 0,C 180,E1 -26166.994,E2 -26166.994} C_VEL
LIN {X 0,Y 108.036,Z 327.026,A -85,B 0,C 180,E1 -26174.913,E2 -26174.913} C_VEL
LIN {X 0,Y 108.302,Z 326.989,A -85,B 0,C 180,E1 -26178.769,E2 -26178.769} C_VEL
LIN {X 0,Y 108.459,Z 326.968,A -85,B 0,C 180,E1 -26186.279,E2 -26186.279} C_VEL
LIN {X 0,Y 108.944,Z 326.914,A -85,B 0,C 180,E1 -26189.994,E2 -26189.994} C_VEL
LIN {X 0,Y 108.335,Z 326.991,A -85,B 0,C 180,E1 -26197.448,E2 -26197.448} C_VEL
LIN {X 0,Y 108.214,Z 327.006,A -85,B 0,C 180,E1 -26203.056,E2 -26203.056} C_VEL
LIN {X 0,Y 108.079,Z 327.017,A -85,B 0,C 180,E1 -26205.672,E2 -26205.672} C_VEL
LIN {X 0,Y 110.014,Z 332.172,A -85,B 0,C 180,E1 -26206.762,E2 -26206.762} C_VEL
LIN {X 0,Y 115.956,Z 346.166,A -85,B 0,C 180,E1 -26209.517,E2 -26209.517} C_VEL
LIN {X 0,Y 123.988,Z 368.084,A -85,B 0,C 180,E1 -26213.148,E2 -26213.148} C_VEL
LIN {X 0,Y 119.595,Z 420.901,A -85,B 0,C 180,E1 -26217.394,E2 -26217.394} C_VEL
LIN {X 0,Y 117.881,Z 435.528,A -85,B 0,C 180,E1 -26219.319,E2 -26219.319} C_VEL
LIN {X 0,Y 115.749,Z 448.583,A -85,B 0,C 180,E1 -26221.787,E2 -26221.787} C_VEL
LIN {X 0,Y 113.635,Z 459.917,A -85,B 0,C 180,E1 -26224.614,E2 -26224.614} C_VEL
LIN {X 0,Y 111.653,Z 469.926,A -85,B 0,C 180,E1 -26227.791,E2 -26227.791} C_VEL
LIN {X 0,Y 109.38,Z 481.173,A -85,B 0,C 180,E1 -26232.364,E2 -26232.364} C_VEL
LIN {X 0,Y 107.554,Z 490.796,A -85,B 0,C 180,E1 -26237.324,E2 -26237.324} C_VEL
LIN {X 0,Y 106.292,Z 498.815,A -85,B 0,C 180,E1 -26242.49,E2 -26242.49} C_VEL
LIN {X 0,Y 105.521,Z 505.478,A -85,B 0,C 180,E1 -26247.806,E2 -26247.806} C_VEL
LIN {X 0,Y 105.317,Z 511.939,A -85,B 0,C 180,E1 -26254.296,E2 -26254.296} C_VEL
LIN {X 0,Y 106.251,Z 516.899,A -85,B 0,C 180,E1 -26260.689,E2 -26260.689} C_VEL
LIN {X 0,Y 108.266,Z 520.58,A -85,B 0,C 180,E1 -26266.783,E2 -26266.783} C_VEL
LIN {X 0,Y 112.906,Z 523.932,A -85,B 0,C 180,E1 -26274.713,E2 -26274.713} C_VEL
LIN {X 0,Y 119.515,Z 525.403,A -85,B 0,C 180,E1 -26281.851,E2 -26281.851} C_VEL
LIN {X 0,Y 127.726,Z 525.039,A -85,B 0,C 180,E1 -26288.009,E2 -26288.009} C_VEL
LIN {X 0,Y 137.165,Z 523.027,A -85,B 0,C 180,E1 -26293.261,E2 -26293.261} C_VEL
LIN {X 0,Y 145.398,Z 520.152,A -85,B 0,C 180,E1 -26296.86,E2 -26296.86} C_VEL
LIN {X 0,Y 154.131,Z 516.14,A -85,B 0,C 180,E1 -26299.999,E2 -26299.999} C_VEL
LIN {X 0,Y 163.441,Z 510.793,A -85,B 0,C 180,E1 -26302.769,E2 -26302.769} C_VEL
LIN {X 0,Y 173.167,Z 503.922,A -85,B 0,C 180,E1 -26305.224,E2 -26305.224} C_VEL
LIN {X 0,Y 181.435,Z 497.004,A -85,B 0,C 180,E1 -26307.03,E2 -26307.03} C_VEL
LIN {X 0,Y 190.154,Z 488.289,A -85,B 0,C 180,E1 -26308.717,E2 -26308.717} C_VEL
LIN {X 0,Y 197.192,Z 479.929,A -85,B 0,C 180,E1 -26309.933,E2 -26309.933} C_VEL
LIN {X 0,Y 196.848,Z 480.442,A -85,B 0,C 180,E1 -26310.319,E2 -26310.319} C_VEL
LIN {X 0,Y 188.169,Z 490.881,A -85,B 0,C 180,E1 -26311.528,E2 -26311.528} C_VEL
LIN {X 0,Y 178.352,Z 500.704,A -85,B 0,C 180,E1 -26313.153,E2 -26313.153} C_VEL
LIN {X 0,Y 167.842,Z 509.47,A -85,B 0,C 180,E1 -26315.277,E2 -26315.277} C_VEL
LIN {X 0,Y 159.189,Z 515.609,A -85,B 0,C 180,E1 -26317.389,E2 -26317.389} C_VEL
LIN {X 0,Y 150.916,Z 520.627,A -85,B 0,C 180,E1 -26319.804,E2 -26319.804} C_VEL
LIN {X 0,Y 142.993,Z 524.695,A -85,B 0,C 180,E1 -26322.516,E2 -26322.516} C_VEL
LIN {X 0,Y 133.388,Z 528.713,A -85,B 0,C 180,E1 -26326.78,E2 -26326.78} C_VEL
LIN {X 0,Y 124.813,Z 531.316,A -85,B 0,C 180,E1 -26331.74,E2 -26331.74} C_VEL
LIN {X 0,Y 117.72,Z 532.603,A -85,B 0,C 180,E1 -26337.51,E2 -26337.51} C_VEL
LIN {X 0,Y 111.987,Z 532.554,A -85,B 0,C 180,E1 -26343.95,E2 -26343.95} C_VEL
LIN {X 0,Y 108.14,Z 531.129,A -85,B 0,C 180,E1 -26351.046,E2 -26351.046} C_VEL
LIN {X 0,Y 106.471,Z 528.389,A -85,B 0,C 180,E1 -26358.586,E2 -26358.586} C_VEL
LIN {X 0,Y 106.372,Z 525.264,A -85,B 0,C 180,E1 -26364.38,E2 -26364.38} C_VEL
LIN {X 0,Y 106.682,Z 522.68,A -85,B 0,C 180,E1 -26368.119,E2 -26368.119} C_VEL
LIN {X 0,Y 106.689,Z 519.432,A -85,B 0,C 180,E1 -26371.893,E2 -26371.893} C_VEL
LIN {X 0,Y 106.68,Z 513.224,A -85,B 0,C 180,E1 -26377.577,E2 -26377.577} C_VEL
LIN {X 0,Y 107.276,Z 505.326,A -85,B 0,C 180,E1 -26383.26,E2 -26383.26} C_VEL
LIN {X 0,Y 108.58,Z 497.258,A -85,B 0,C 180,E1 -26387.91,E2 -26387.91} C_VEL
LIN {X 0,Y 110.376,Z 487.363,A -85,B 0,C 180,E1 -26392.464,E2 -26392.464} C_VEL
LIN {X 0,Y 112.622,Z 476.349,A -85,B 0,C 180,E1 -26396.403,E2 -26396.403} C_VEL
LIN {X 0,Y 114.986,Z 464.105,A -85,B 0,C 180,E1 -26399.779,E2 -26399.779} C_VEL
LIN {X 0,Y 117.273,Z 451.207,A -85,B 0,C 180,E1 -26402.388,E2 -26402.388} C_VEL
LIN {X 0,Y 119.094,Z 438.047,A -85,B 0,C 180,E1 -26404.313,E2 -26404.313} C_VEL
LIN {X 0,Y 120.017,Z 427.539,A -85,B 0,C 180,E1 -26405.386,E2 -26405.386} C_VEL
LIN {X 0,Y 119.916,Z 421.76,A -85,B 0,C 180,E1 -26405.965,E2 -26405.965} C_VEL
LIN {X 0,Y 115.919,Z 402.903,A -85,B 0,C 180,E1 -26408.297,E2 -26408.297} C_VEL
LIN {X 0,Y 115.742,Z 397.101,A -85,B 0,C 180,E1 -26408.878,E2 -26408.878} C_VEL
LIN {X 0,Y 115.972,Z 391.325,A -85,B 0,C 180,E1 -26409.401,E2 -26409.401} C_VEL
LIN {X 0,Y 114.462,Z 368.432,A -85,B 0,C 180,E1 -26411.924,E2 -26411.924} C_VEL
LIN {X 0,Y 108.584,Z 348.102,A -85,B 0,C 180,E1 -26415.276,E2 -26415.276} C_VEL
LIN {X 0,Y 105.098,Z 338.054,A -85,B 0,C 180,E1 -26417.217,E2 -26417.217} C_VEL
LIN {X 0,Y 100.73,Z 328.465,A -85,B 0,C 180,E1 -26419.532,E2 -26419.532} C_VEL
LIN {X 0,Y 100.625,Z 327.952,A -85,B 0,C 180,E1 -26419.66,E2 -26419.66} C_VEL
LIN {X 0,Y 100.689,Z 327.942,A -85,B 0,C 180,E1 -26426.889,E2 -26426.889} C_VEL
LIN {X 0,Y 100.746,Z 327.932,A -85,B 0,C 180,E1 -26435.254,E2 -26435.254} C_VEL
LIN {X 0,Y 100.777,Z 327.931,A -85,B 0,C 180,E1 -26439.591,E2 -26439.591} C_VEL
LIN {X 0,Y 101.113,Z 327.889,A -85,B 0,C 180,E1 -26447.962,E2 -26447.962} C_VEL
LIN {X 0,Y 101.22,Z 327.873,A -85,B 0,C 180,E1 -26452.016,E2 -26452.016} C_VEL
LIN {X 0,Y 101.834,Z 327.797,A -85,B 0,C 180,E1 -26459.998,E2 -26459.998} C_VEL
LIN {X 0,Y 101.218,Z 327.875,A -85,B 0,C 180,E1 -26467.98,E2 -26467.98} C_VEL
LIN {X 0,Y 101.048,Z 327.896,A -85,B 0,C 180,E1 -26473.162,E2 -26473.162} C_VEL
LIN {X 0,Y 100.779,Z 327.927,A -85,B 0,C 180,E1 -26480.405,E2 -26480.405} C_VEL
LIN {X 0,Y 100.734,Z 327.936,A -85,B 0,C 180,E1 -26484.906,E2 -26484.906} C_VEL
LIN {X 0,Y 100.687,Z 327.942,A -85,B 0,C 180,E1 -26493.109,E2 -26493.109} C_VEL
LIN {X 0,Y 100.639,Z 327.949,A -85,B 0,C 180,E1 -26499.807,E2 -26499.807} C_VEL
LIN {X 0,Y 100.661,Z 327.941,A -85,B 0,C 180,E1 -26505.715,E2 -26505.715} C_VEL
LIN {X 0,Y 100.662,Z 327.943,A -85,B 0,C 180,E1 -26511.067,E2 -26511.067} C_VEL
LIN {X 0,Y 100.7,Z 327.941,A -85,B 0,C 180,E1 -26516.873,E2 -26516.873} C_VEL
LIN {X 0,Y 100.786,Z 327.93,A -85,B 0,C 180,E1 -26525.263,E2 -26525.263} C_VEL
LIN {X 0,Y 100.816,Z 327.919,A -85,B 0,C 180,E1 -26529.596,E2 -26529.596} C_VEL
LIN {X 0,Y 101.196,Z 327.872,A -85,B 0,C 180,E1 -26537.969,E2 -26537.969} C_VEL
LIN {X 0,Y 101.275,Z 327.87,A -85,B 0,C 180,E1 -26542.017,E2 -26542.017} C_VEL
LIN {X 0,Y 101.868,Z 327.795,A -85,B 0,C 180,E1 -26549.994,E2 -26549.994} C_VEL
LIN {X 0,Y 101.276,Z 327.87,A -85,B 0,C 180,E1 -26557.971,E2 -26557.971} C_VEL
LIN {X 0,Y 101.122,Z 327.889,A -85,B 0,C 180,E1 -26563.814,E2 -26563.814} C_VEL
LIN {X 0,Y 102.106,Z 330.812,A -85,B 0,C 180,E1 -26564.51,E2 -26564.51} C_VEL
LIN {X 0,Y 108.269,Z 345.283,A -85,B 0,C 180,E1 -26567.736,E2 -26567.736} C_VEL
LIN {X 0,Y 115.37,Z 364.145,A -85,B 0,C 180,E1 -26571.172,E2 -26571.172} C_VEL
LIN {X 0,Y 117.255,Z 369.7,A -85,B 0,C 180,E1 -26572.085,E2 -26572.085} C_VEL
LIN {X 0,Y 112.834,Z 420.45,A -85,B 0,C 180,E1 -26576.361,E2 -26576.361} C_VEL
LIN {X 0,Y 111.212,Z 433.939,A -85,B 0,C 180,E1 -26578.188,E2 -26578.188} C_VEL
LIN {X 0,Y 109.189,Z 446.551,A -85,B 0,C 180,E1 -26580.58,E2 -26580.58} C_VEL
LIN {X 0,Y 106.765,Z 459.052,A -85,B 0,C 180,E1 -26583.795,E2 -26583.795} C_VEL
LIN {X 0,Y 104.468,Z 470.189,A -85,B 0,C 180,E1 -26587.518,E2 -26587.518} C_VEL
LIN {X 0,Y 102.38,Z 480.471,A -85,B 0,C 180,E1 -26591.912,E2 -26591.912} C_VEL
LIN {X 0,Y 100.521,Z 489.969,A -85,B 0,C 180,E1 -26597.028,E2 -26597.028} C_VEL
LIN {X 0,Y 99.144,Z 499.025,A -85,B 0,C 180,E1 -26603.159,E2 -26603.159} C_VEL
LIN {X 0,Y 98.389,Z 505.795,A -85,B 0,C 180,E1 -26608.978,E2 -26608.978} C_VEL
LIN {X 0,Y 98.287,Z 511.106,A -85,B 0,C 180,E1 -26614.596,E2 -26614.596} C_VEL
LIN {X 0,Y 99.317,Z 516.367,A -85,B 0,C 180,E1 -26621.434,E2 -26621.434} C_VEL
LIN {X 0,Y 101.519,Z 520.351,A -85,B 0,C 180,E1 -26628.015,E2 -26628.015} C_VEL
LIN {X 0,Y 105.75,Z 523.602,A -85,B 0,C 180,E1 -26635.326,E2 -26635.326} C_VEL
LIN {X 0,Y 109.672,Z 525.068,A -85,B 0,C 180,E1 -26640.002,E2 -26640.002} C_VEL
LIN {X 0,Y 113.336,Z 525.731,A -85,B 0,C 180,E1 -26643.557,E2 -26643.557} C_VEL
LIN {X 0,Y 121.039,Z 525.865,A -85,B 0,C 180,E1 -26649.288,E2 -26649.288} C_VEL
LIN {X 0,Y 130.752,Z 524.426,A -85,B 0,C 180,E1 -26654.686,E2 -26654.686} C_VEL
LIN {X 0,Y 137.804,Z 522.534,A -85,B 0,C 180,E1 -26657.82,E2 -26657.82} C_VEL
LIN {X 0,Y 146.768,Z 519.258,A -85,B 0,C 180,E1 -26661.049,E2 -26661.049} C_VEL
LIN {X 0,Y 156.265,Z 514.703,A -85,B 0,C 180,E1 -26663.878,E2 -26663.878} C_VEL
LIN {X 0,Y 166.753,Z 508.412,A -85,B 0,C 180,E1 -26666.49,E2 -26666.49} C_VEL
LIN {X 0,Y 176.506,Z 501.254,A -85,B 0,C 180,E1 -26668.544,E2 -26668.544} C_VEL
LIN {X 0,Y 183.536,Z 495.109,A -85,B 0,C 180,E1 -26669.856,E2 -26669.856} C_VEL
LIN {X 0,Y 173.114,Z 504.448,A -85,B 0,C 180,E1 -26671.527,E2 -26671.527} C_VEL
LIN {X 0,Y 163.932,Z 511.326,A -85,B 0,C 180,E1 -26673.297,E2 -26673.297} C_VEL
LIN {X 0,Y 152.138,Z 518.633,A -85,B 0,C 180,E1 -26676.074,E2 -26676.074} C_VEL
LIN {X 0,Y 141.026,Z 524.225,A -85,B 0,C 180,E1 -26679.441,E2 -26679.441} C_VEL
LIN {X 0,Y 133.201,Z 527.33,A -85,B 0,C 180,E1 -26682.395,E2 -26682.395} C_VEL
LIN {X 0,Y 123.667,Z 530.296,A -85,B 0,C 180,E1 -26687.016,E2 -26687.016} C_VEL
LIN {X 0,Y 115.361,Z 531.869,A -85,B 0,C 180,E1 -26692.479,E2 -26692.479} C_VEL
LIN {X 0,Y 108.467,Z 532.14,A -85,B 0,C 180,E1 -26698.789,E2 -26698.789} C_VEL
LIN {X 0,Y 103.271,Z 531.117,A -85,B 0,C 180,E1 -26705.91,E2 -26705.91} C_VEL
LIN {X 0,Y 100.266,Z 528.786,A -85,B 0,C 180,E1 -26713.726,E2 -26713.726} C_VEL
LIN {X 0,Y 99.392,Z 524.987,A -85,B 0,C 180,E1 -26721.877,E2 -26721.877} C_VEL
LIN {X 0,Y 99.773,Z 521.042,A -85,B 0,C 180,E1 -26727.988,E2 -26727.988} C_VEL
LIN {X 0,Y 99.737,Z 517.539,A -85,B 0,C 180,E1 -26732.025,E2 -26732.025} C_VEL
LIN {X 0,Y 99.716,Z 512.187,A -85,B 0,C 180,E1 -26737.091,E2 -26737.091} C_VEL
LIN {X 0,Y 100.285,Z 504.178,A -85,B 0,C 180,E1 -26743.17,E2 -26743.17} C_VEL
LIN {X 0,Y 101.596,Z 496.025,A -85,B 0,C 180,E1 -26748.142,E2 -26748.142} C_VEL
LIN {X 0,Y 103.48,Z 485.997,A -85,B 0,C 180,E1 -26752.991,E2 -26752.991} C_VEL
LIN {X 0,Y 105.789,Z 474.867,A -85,B 0,C 180,E1 -26757.18,E2 -26757.18} C_VEL
LIN {X 0,Y 107.939,Z 464.123,A -85,B 0,C 180,E1 -26760.309,E2 -26760.309} C_VEL
LIN {X 0,Y 110.259,Z 451.363,A -85,B 0,C 180,E1 -26763.081,E2 -26763.081} C_VEL
LIN {X 0,Y 112.256,Z 437.582,A -85,B 0,C 180,E1 -26765.221,E2 -26765.221} C_VEL
LIN {X 0,Y 113.76,Z 421.01,A -85,B 0,C 180,E1 -26766.862,E2 -26766.862} C_VEL
LIN {X 0,Y 115.742,Z 397.101,A -85,B 0,C 180,E1 -26768.878,E2 -26768.878} C_VEL
LIN {X 0,Y 115.469,Z 391.364,A -85,B 0,C 180,E1 -26769.485,E2 -26769.485} C_VEL
LIN {X 0,Y 114.094,Z 385.829,A -85,B 0,C 180,E1 -26770.274,E2 -26770.274} C_VEL
LIN {X 0,Y 107.342,Z 367.864,A -85,B 0,C 180,E1 -26773.437,E2 -26773.437} C_VEL
LIN {X 0,Y 101.219,Z 347.044,A -85,B 0,C 180,E1 -26777.22,E2 -26777.22} C_VEL
LIN {X 0,Y 98.806,Z 340.369,A -85,B 0,C 180,E1 -26778.685,E2 -26778.685} C_VEL
LIN {X 0,Y 93.707,Z 329.645,A -85,B 0,C 180,E1 -26781.602,E2 -26781.602} C_VEL
LIN {X 0,Y 93.532,Z 328.832,A -85,B 0,C 180,E1 -26781.859,E2 -26781.859} C_VEL
